LIN {X 0,Y 351.097,Z 362.91,A -85,B 0,C 180,E1 -17556.898,E2 -17556.898} C_VEL
LIN {X 0,Y 348.285,Z 360.251,A -85,B 0,C 180,E1 -17558.664,E2 -17558.664} C_VEL
LIN {X 0,Y 346.12,Z 358.177,A -85,B 0,C 180,E1 -17559.821,E2 -17559.821} C_VEL
LIN {X 0,Y 342.771,Z 355.678,A -85,B 0,C 180,E1 -17561.154,E2 -17561.154} C_VEL
LIN {X 0,Y 338.579,Z 351.959,A -85,B 0,C 180,E1 -17562.731,E2 -17562.731} C_VEL
LIN {X 0,Y 335.792,Z 349.388,A -85,B 0,C 180,E1 -17563.695,E2 -17563.695} C_VEL
LIN {X 0,Y 331.401,Z 345.387,A -85,B 0,C 180,E1 -17565.057,E2 -17565.057} C_VEL
LIN {X 0,Y 325.553,Z 339.743,A -85,B 0,C 180,E1 -17566.706,E2 -17566.706} C_VEL
LIN {X 0,Y 318.538,Z 332.574,A -85,B 0,C 180,E1 -17568.462,E2 -17568.462} C_VEL
LIN {X 0,Y 312.151,Z 325.702,A -85,B 0,C 180,E1 -17569.9,E2 -17569.9} C_VEL
LIN {X 0,Y 303.087,Z 315.131,A -85,B 0,C 180,E1 -17571.777,E2 -17571.777} C_VEL
LIN {X 0,Y 294.903,Z 304.725,A -85,B 0,C 180,E1 -17573.408,E2 -17573.408} C_VEL
LIN {X 0,Y 288.383,Z 294.709,A -85,B 0,C 180,E1 -17574.719,E2 -17574.719} C_VEL
LIN {X 0,Y 283.758,Z 285.694,A -85,B 0,C 180,E1 -17575.657,E2 -17575.657} C_VEL
LIN {X 0,Y 277.541,Z 272.57,A -85,B 0,C 180,E1 -17576.757,E2 -17576.757} C_VEL
LIN {X 0,Y 277.287,Z 271.445,A -85,B 0,C 180,E1 -17576.818,E2 -17576.818} C_VEL
LIN {X 0,Y 277.223,Z 271.454,A -85,B 0,C 180,E1 -17580.487,E2 -17580.487} C_VEL
LIN {X 0,Y 277.2,Z 271.458,A -85,B 0,C 180,E1 -17583.902,E2 -17583.902} C_VEL
LIN {X 0,Y 277.232,Z 271.452,A -85,B 0,C 180,E1 -17587.474,E2 -17587.474} C_VEL
LIN {X 0,Y 277.222,Z 271.452,A -85,B 0,C 180,E1 -17591.233,E2 -17591.233} C_VEL
LIN {X 0,Y 277.247,Z 271.449,A -85,B 0,C 180,E1 -17595.216,E2 -17595.216} C_VEL
LIN {X 0,Y 277.258,Z 271.45,A -85,B 0,C 180,E1 -17599.502,E2 -17599.502} C_VEL
LIN {X 0,Y 277.25,Z 271.448,A -85,B 0,C 180,E1 -17602.541,E2 -17602.541} C_VEL
LIN {X 0,Y 277.222,Z 271.451,A -85,B 0,C 180,E1 -17606.113,E2 -17606.113} C_VEL
LIN {X 0,Y 277.233,Z 271.452,A -85,B 0,C 180,E1 -17609.547,E2 -17609.547} C_VEL
LIN {X 0,Y 277.329,Z 271.44,A -85,B 0,C 180,E1 -17612.872,E2 -17612.872} C_VEL
LIN {X 0,Y 277.272,Z 271.443,A -85,B 0,C 180,E1 -17616.085,E2 -17616.085} C_VEL
LIN {X 0,Y 277.297,Z 271.441,A -85,B 0,C 180,E1 -17620.773,E2 -17620.773} C_VEL
LIN {X 0,Y 277.393,Z 271.428,A -85,B 0,C 180,E1 -17625.333,E2 -17625.333} C_VEL
LIN {X 0,Y 277.444,Z 271.421,A -85,B 0,C 180,E1 -17629.796,E2 -17629.796} C_VEL
LIN {X 0,Y 277.604,Z 271.406,A -85,B 0,C 180,E1 -17632.737,E2 -17632.737} C_VEL
LIN {X 0,Y 277.799,Z 271.368,A -85,B 0,C 180,E1 -17638.559,E2 -17638.559} C_VEL
LIN {X 0,Y 277.806,Z 271.376,A -85,B 0,C 180,E1 -17641.458,E2 -17641.458} C_VEL
LIN {X 0,Y 277.598,Z 271.404,A -85,B 0,C 180,E1 -17647.28,E2 -17647.28} C_VEL
LIN {X 0,Y 277.455,Z 271.425,A -85,B 0,C 180,E1 -17650.221,E2 -17650.221} C_VEL
LIN {X 0,Y 277.375,Z 271.433,A -85,B 0,C 180,E1 -17654.685,E2 -17654.685} C_VEL
LIN {X 0,Y 277.283,Z 271.445,A -85,B 0,C 180,E1 -17659.246,E2 -17659.246} C_VEL
LIN {X 0,Y 277.263,Z 271.448,A -85,B 0,C 180,E1 -17663.934,E2 -17663.934} C_VEL
LIN {X 0,Y 277.221,Z 271.451,A -85,B 0,C 180,E1 -17666.268,E2 -17666.268} C_VEL
LIN {X 0,Y 276.55,Z 271.54,A -85,B 0,C 180,E1 -17667.481,E2 -17667.481} C_VEL
LIN {X 0,Y 273.663,Z 271.899,A -85,B 0,C 180,E1 -17669.456,E2 -17669.456} C_VEL
LIN {X 0,Y 271.269,Z 272.403,A -85,B 0,C 180,E1 -17671.059,E2 -17671.059} C_VEL
LIN {X 0,Y 270.324,Z 272.925,A -85,B 0,C 180,E1 -17672.299,E2 -17672.299} C_VEL
LIN {X 0,Y 270.291,Z 273.131,A -85,B 0,C 180,E1 -17672.718,E2 -17672.718} C_VEL
LIN {X 0,Y 270.597,Z 275.334,A -85,B 0,C 180,E1 -17676.689,E2 -17676.689} C_VEL
LIN {X 0,Y 271.058,Z 278.164,A -85,B 0,C 180,E1 -17681.245,E2 -17681.245} C_VEL
LIN {X 0,Y 271.419,Z 281.232,A -85,B 0,C 180,E1 -17685.644,E2 -17685.644} C_VEL
LIN {X 0,Y 271.327,Z 283.569,A -85,B 0,C 180,E1 -17688.701,E2 -17688.701} C_VEL
LIN {X 0,Y 270.949,Z 285.847,A -85,B 0,C 180,E1 -17691.5,E2 -17691.5} C_VEL
LIN {X 0,Y 270.368,Z 288.968,A -85,B 0,C 180,E1 -17695.12,E2 -17695.12} C_VEL
LIN {X 0,Y 269.734,Z 292.721,A -85,B 0,C 180,E1 -17699.308,E2 -17699.308} C_VEL
LIN {X 0,Y 269.233,Z 295.826,A -85,B 0,C 180,E1 -17702.634,E2 -17702.634} C_VEL
LIN {X 0,Y 270.907,Z 301.981,A -85,B 0,C 180,E1 -17703.108,E2 -17703.108} C_VEL
LIN {X 0,Y 273.793,Z 313.364,A -85,B 0,C 180,E1 -17704.128,E2 -17704.128} C_VEL
LIN {X 0,Y 275.705,Z 322.952,A -85,B 0,C 180,E1 -17705.113,E2 -17705.113} C_VEL
LIN {X 0,Y 277,Z 333.021,A -85,B 0,C 180,E1 -17706.288,E2 -17706.288} C_VEL
LIN {X 0,Y 277.683,Z 342.384,A -85,B 0,C 180,E1 -17707.542,E2 -17707.542} C_VEL
LIN {X 0,Y 277.852,Z 346.126,A -85,B 0,C 180,E1 -17708.094,E2 -17708.094} C_VEL
LIN {X 0,Y 275.725,Z 357.626,A -85,B 0,C 180,E1 -17709.873,E2 -17709.873} C_VEL
LIN {X 0,Y 274.037,Z 366.483,A -85,B 0,C 180,E1 -17711.622,E2 -17711.622} C_VEL
LIN {X 0,Y 272.809,Z 372.974,A -85,B 0,C 180,E1 -17713.153,E2 -17713.153} C_VEL
LIN {X 0,Y 271.496,Z 379.514,A -85,B 0,C 180,E1 -17714.998,E2 -17714.998} C_VEL
LIN {X 0,Y 270.527,Z 384.016,A -85,B 0,C 180,E1 -17716.479,E2 -17716.479} C_VEL
LIN {X 0,Y 269.512,Z 389.513,A -85,B 0,C 180,E1 -17718.722,E2 -17718.722} C_VEL
LIN {X 0,Y 268.8,Z 393.843,A -85,B 0,C 180,E1 -17720.975,E2 -17720.975} C_VEL
LIN {X 0,Y 268.481,Z 396.213,A -85,B 0,C 180,E1 -17722.479,E2 -17722.479} C_VEL
LIN {X 0,Y 268.229,Z 398.793,A -85,B 0,C 180,E1 -17724.713,E2 -17724.713} C_VEL
LIN {X 0,Y 268.184,Z 400.47,A -85,B 0,C 180,E1 -17726.996,E2 -17726.996} C_VEL
LIN {X 0,Y 268.192,Z 401.061,A -85,B 0,C 180,E1 -17728.498,E2 -17728.498} C_VEL
LIN {X 0,Y 268.192,Z 401.061,A -85,B 0,C 180,E1 -17731.502,E2 -17731.502} C_VEL
LIN {X 0,Y 268.184,Z 400.47,A -85,B 0,C 180,E1 -17733.004,E2 -17733.004} C_VEL
LIN {X 0,Y 268.31,Z 398.017,A -85,B 0,C 180,E1 -17736.014,E2 -17736.014} C_VEL
LIN {X 0,Y 268.618,Z 395.061,A -85,B 0,C 180,E1 -17738.273,E2 -17738.273} C_VEL
LIN {X 0,Y 269.258,Z 391.069,A -85,B 0,C 180,E1 -17740.527,E2 -17740.527} C_VEL
LIN {X 0,Y 270.136,Z 385.933,A -85,B 0,C 180,E1 -17742.776,E2 -17742.776} C_VEL
LIN {X 0,Y 271.233,Z 380.67,A -85,B 0,C 180,E1 -17744.633,E2 -17744.633} C_VEL
LIN {X 0,Y 272.49,Z 374.349,A -85,B 0,C 180,E1 -17746.481,E2 -17746.481} C_VEL
LIN {X 0,Y 273.898,Z 367.698,A -85,B 0,C 180,E1 -17748.099,E2 -17748.099} C_VEL
LIN {X 0,Y 275.325,Z 359.545,A -85,B 0,C 180,E1 -17749.768,E2 -17749.768} C_VEL
LIN {X 0,Y 276.982,Z 351.016,A -85,B 0,C 180,E1 -17751.196,E2 -17751.196} C_VEL
LIN {X 0,Y 277.855,Z 346.126,A -85,B 0,C 180,E1 -17751.905,E2 -17751.905} C_VEL
LIN {X 0,Y 277.327,Z 336.813,A -85,B 0,C 180,E1 -17753.227,E2 -17753.227} C_VEL
LIN {X 0,Y 276.285,Z 326.665,A -85,B 0,C 180,E1 -17754.465,E2 -17754.465} C_VEL
LIN {X 0,Y 274.542,Z 316.92,A -85,B 0,C 180,E1 -17755.519,E2 -17755.519} C_VEL
LIN {X 0,Y 272.191,Z 306.812,A -85,B 0,C 180,E1 -17756.473,E2 -17756.473} C_VEL
LIN {X 0,Y 269.34,Z 296.803,A -85,B 0,C 180,E1 -17757.293,E2 -17757.293} C_VEL
LIN {X 0,Y 269.233,Z 295.84,A -85,B 0,C 180,E1 -17757.351,E2 -17757.351} C_VEL
LIN {X 0,Y 269.789,Z 292.071,A -85,B 0,C 180,E1 -17761.399,E2 -17761.399} C_VEL
LIN {X 0,Y 270.376,Z 288.938,A -85,B 0,C 180,E1 -17764.879,E2 -17764.879} C_VEL
LIN {X 0,Y 271.024,Z 285.471,A -85,B 0,C 180,E1 -17768.918,E2 -17768.918} C_VEL
LIN {X 0,Y 271.38,Z 282.742,A -85,B 0,C 180,E1 -17772.324,E2 -17772.324} C_VEL
LIN {X 0,Y 271.423,Z 281.192,A -85,B 0,C 180,E1 -17774.355,E2 -17774.355} C_VEL
LIN {X 0,Y 271.058,Z 278.155,A -85,B 0,C 180,E1 -17778.755,E2 -17778.755} C_VEL
LIN {X 0,Y 270.59,Z 275.327,A -85,B 0,C 180,E1 -17783.31,E2 -17783.31} C_VEL
LIN {X 0,Y 270.343,Z 273.321,A -85,B 0,C 180,E1 -17786.904,E2 -17786.904} C_VEL
LIN {X 0,Y 270.187,Z 272.33,A -85,B 0,C 180,E1 -17789.134,E2 -17789.134} C_VEL
LIN {X 0,Y 270.198,Z 272.33,A -85,B 0,C 180,E1 -17792.171,E2 -17792.171} C_VEL
LIN {X 0,Y 270.191,Z 272.331,A -85,B 0,C 180,E1 -17795.557,E2 -17795.557} C_VEL
LIN {X 0,Y 270.226,Z 272.328,A -85,B 0,C 180,E1 -17800.231,E2 -17800.231} C_VEL
LIN {X 0,Y 270.342,Z 272.309,A -85,B 0,C 180,E1 -17804.924,E2 -17804.924} C_VEL
LIN {X 0,Y 270.387,Z 272.304,A -85,B 0,C 180,E1 -17809.509,E2 -17809.509} C_VEL
LIN {X 0,Y 270.561,Z 272.281,A -85,B 0,C 180,E1 -17812.529,E2 -17812.529} C_VEL
LIN {X 0,Y 270.77,Z 272.253,A -85,B 0,C 180,E1 -17818.504,E2 -17818.504} C_VEL
LIN {X 0,Y 270.765,Z 272.242,A -85,B 0,C 180,E1 -17821.479,E2 -17821.479} C_VEL
LIN {X 0,Y 270.563,Z 272.285,A -85,B 0,C 180,E1 -17827.453,E2 -17827.453} C_VEL
LIN {X 0,Y 270.397,Z 272.299,A -85,B 0,C 180,E1 -17830.473,E2 -17830.473} C_VEL
LIN {X 0,Y 270.351,Z 272.306,A -85,B 0,C 180,E1 -17835.058,E2 -17835.058} C_VEL
LIN {X 0,Y 270.237,Z 272.317,A -85,B 0,C 180,E1 -17839.75,E2 -17839.75} C_VEL
LIN {X 0,Y 270.213,Z 272.325,A -85,B 0,C 180,E1 -17844.58,E2 -17844.58} C_VEL
LIN {X 0,Y 270.245,Z 272.32,A -85,B 0,C 180,E1 -17847.9,E2 -17847.9} C_VEL
LIN {X 0,Y 270.154,Z 272.332,A -85,B 0,C 180,E1 -17851.34,E2 -17851.34} C_VEL
LIN {X 0,Y 270.182,Z 272.33,A -85,B 0,C 180,E1 -17854.895,E2 -17854.895} C_VEL
LIN {X 0,Y 270.188,Z 272.331,A -85,B 0,C 180,E1 -17858.709,E2 -17858.709} C_VEL
LIN {X 0,Y 270.192,Z 272.329,A -85,B 0,C 180,E1 -17862.539,E2 -17862.539} C_VEL
LIN {X 0,Y 270.191,Z 272.328,A -85,B 0,C 180,E1 -17866.729,E2 -17866.729} C_VEL
LIN {X 0,Y 270.203,Z 272.325,A -85,B 0,C 180,E1 -17869.44,E2 -17869.44} C_VEL
LIN {X 0,Y 270.198,Z 272.328,A -85,B 0,C 180,E1 -17873.719,E2 -17873.719} C_VEL
LIN {X 0,Y 270.155,Z 272.332,A -85,B 0,C 180,E1 -17876.887,E2 -17876.887} C_VEL
LIN {X 0,Y 270.147,Z 272.335,A -85,B 0,C 180,E1 -17880.377,E2 -17880.377} C_VEL
LIN {X 0,Y 270.244,Z 272.323,A -85,B 0,C 180,E1 -17882.432,E2 -17882.432} C_VEL
LIN {X 0,Y 271.191,Z 275.041,A -85,B 0,C 180,E1 -17882.63,E2 -17882.63} C_VEL
LIN {X 0,Y 277.134,Z 287.397,A -85,B 0,C 180,E1 -17883.752,E2 -17883.752} C_VEL
LIN {X 0,Y 281.702,Z 297.031,A -85,B 0,C 180,E1 -17884.796,E2 -17884.796} C_VEL
LIN {X 0,Y 287.454,Z 306.253,A -85,B 0,C 180,E1 -17886.06,E2 -17886.06} C_VEL
LIN {X 0,Y 294.959,Z 316.48,A -85,B 0,C 180,E1 -17887.706,E2 -17887.706} C_VEL
LIN {X 0,Y 304.263,Z 327.414,A -85,B 0,C 180,E1 -17889.728,E2 -17889.728} C_VEL
LIN {X 0,Y 312.75,Z 336.664,A -85,B 0,C 180,E1 -17891.664,E2 -17891.664} C_VEL
LIN {X 0,Y 318.182,Z 342.223,A -85,B 0,C 180,E1 -17893.002,E2 -17893.002} C_VEL
LIN {X 0,Y 324.333,Z 348.16,A -85,B 0,C 180,E1 -17894.656,E2 -17894.656} C_VEL
LIN {X 0,Y 330.14,Z 353.561,A -85,B 0,C 180,E1 -17896.458,E2 -17896.458} C_VEL
LIN {X 0,Y 334.126,Z 357.349,A -85,B 0,C 180,E1 -17897.858,E2 -17897.858} C_VEL
LIN {X 0,Y 338.742,Z 361.057,A -85,B 0,C 180,E1 -17899.606,E2 -17899.606} C_VEL
LIN {X 0,Y 341.574,Z 363.402,A -85,B 0,C 180,E1 -17900.908,E2 -17900.908} C_VEL
LIN {X 0,Y 345.018,Z 366.712,A -85,B 0,C 180,E1 -17902.98,E2 -17902.98} C_VEL
LIN {X 0,Y 346.829,Z 368.073,A -85,B 0,C 180,E1 -17904.185,E2 -17904.185} C_VEL
LIN {X 0,Y 348.425,Z 369.044,A -85,B 0,C 180,E1 -17905.372,E2 -17905.372} C_VEL
LIN {X 0,Y 349.812,Z 369.646,A -85,B 0,C 180,E1 -17906.545,E2 -17906.545} C_VEL
LIN {X 0,Y 350.894,Z 370,A -85,B 0,C 180,E1 -17907.704,E2 -17907.704} C_VEL
LIN {X 0,Y 351.655,Z 370.14,A -85,B 0,C 180,E1 -17908.855,E2 -17908.855} C_VEL
LIN {X 0,Y 351.924,Z 370.171,A -85,B 0,C 180,E1 -17910,E2 -17910} C_VEL
LIN {X 0,Y 351.449,Z 370.117,A -85,B 0,C 180,E1 -17911.444,E2 -17911.444} C_VEL
LIN {X 0,Y 350.893,Z 369.986,A -85,B 0,C 180,E1 -17912.296,E2 -17912.296} C_VEL
LIN {X 0,Y 349.809,Z 369.639,A -85,B 0,C 180,E1 -17913.455,E2 -17913.455} C_VEL
LIN {X 0,Y 348.421,Z 369.058,A -85,B 0,C 180,E1 -17914.628,E2 -17914.628} C_VEL
LIN {X 0,Y 346.308,Z 367.73,A -85,B 0,C 180,E1 -17916.158,E2 -17916.158} C_VEL
LIN {X 0,Y 343.076,Z 364.884,A -85,B 0,C 180,E1 -17918.244,E2 -17918.244} C_VEL
LIN {X 0,Y 340.826,Z 362.661,A -85,B 0,C 180,E1 -17919.495,E2 -17919.495} C_VEL
LIN {X 0,Y 336.651,Z 359.474,A -85,B 0,C 180,E1 -17921.187,E2 -17921.187} C_VEL
LIN {X 0,Y 331.755,Z 355.007,A -85,B 0,C 180,E1 -17923.019,E2 -17923.019} C_VEL
LIN {X 0,Y 326.763,Z 350.61,A -85,B 0,C 180,E1 -17924.608,E2 -17924.608} C_VEL
LIN {X 0,Y 321.747,Z 345.628,A -85,B 0,C 180,E1 -17926.072,E2 -17926.072} C_VEL
LIN {X 0,Y 315.363,Z 339.315,A -85,B 0,C 180,E1 -17927.729,E2 -17927.729} C_VEL
LIN {X 0,Y 309.544,Z 333.151,A -85,B 0,C 180,E1 -17929.091,E2 -17929.091} C_VEL
LIN {X 0,Y 301.027,Z 323.692,A -85,B 0,C 180,E1 -17930.985,E2 -17930.985} C_VEL
LIN {X 0,Y 291.898,Z 312.497,A -85,B 0,C 180,E1 -17932.964,E2 -17932.964} C_VEL
LIN {X 0,Y 285.429,Z 303.26,A -85,B 0,C 180,E1 -17934.379,E2 -17934.379} C_VEL
LIN {X 0,Y 279.999,Z 293.639,A -85,B 0,C 180,E1 -17935.6,E2 -17935.6} C_VEL
LIN {X 0,Y 273.951,Z 280.6,A -85,B 0,C 180,E1 -17936.882,E2 -17936.882} C_VEL
LIN {X 0,Y 270.431,Z 273.312,A -85,B 0,C 180,E1 -17937.505,E2 -17937.505} C_VEL
LIN {X 0,Y 270.232,Z 272.325,A -85,B 0,C 180,E1 -17937.598,E2 -17937.598} C_VEL
LIN {X 0,Y 270.136,Z 272.335,A -85,B 0,C 180,E1 -17941.354,E2 -17941.354} C_VEL
LIN {X 0,Y 270.156,Z 272.332,A -85,B 0,C 180,E1 -17944.911,E2 -17944.911} C_VEL
LIN {X 0,Y 270.179,Z 272.329,A -85,B 0,C 180,E1 -17948.724,E2 -17948.724} C_VEL
LIN {X 0,Y 270.188,Z 272.327,A -85,B 0,C 180,E1 -17952.554,E2 -17952.554} C_VEL
LIN {X 0,Y 270.193,Z 272.327,A -85,B 0,C 180,E1 -17956.744,E2 -17956.744} C_VEL
LIN {X 0,Y 270.21,Z 272.327,A -85,B 0,C 180,E1 -17959.455,E2 -17959.455} C_VEL
LIN {X 0,Y 270.222,Z 272.325,A -85,B 0,C 180,E1 -17963.73,E2 -17963.73} C_VEL
LIN {X 0,Y 270.173,Z 272.33,A -85,B 0,C 180,E1 -17966.901,E2 -17966.901} C_VEL
LIN {X 0,Y 270.199,Z 272.326,A -85,B 0,C 180,E1 -17970.395,E2 -17970.395} C_VEL
LIN {X 0,Y 270.233,Z 272.32,A -85,B 0,C 180,E1 -17973.772,E2 -17973.772} C_VEL
LIN {X 0,Y 270.186,Z 272.331,A -85,B 0,C 180,E1 -17977.045,E2 -17977.045} C_VEL
LIN {X 0,Y 270.237,Z 272.317,A -85,B 0,C 180,E1 -17980.25,E2 -17980.25} C_VEL
LIN {X 0,Y 270.351,Z 272.306,A -85,B 0,C 180,E1 -17984.942,E2 -17984.942} C_VEL
LIN {X 0,Y 270.397,Z 272.299,A -85,B 0,C 180,E1 -17989.527,E2 -17989.527} C_VEL
LIN {X 0,Y 270.563,Z 272.285,A -85,B 0,C 180,E1 -17992.547,E2 -17992.547} C_VEL
LIN {X 0,Y 270.765,Z 272.242,A -85,B 0,C 180,E1 -17998.521,E2 -17998.521} C_VEL
LIN {X 0,Y 270.77,Z 272.253,A -85,B 0,C 180,E1 -18001.496,E2 -18001.496} C_VEL
LIN {X 0,Y 270.561,Z 272.282,A -85,B 0,C 180,E1 -18007.471,E2 -18007.471} C_VEL
LIN {X 0,Y 270.387,Z 272.304,A -85,B 0,C 180,E1 -18010.491,E2 -18010.491} C_VEL
LIN {X 0,Y 270.342,Z 272.309,A -85,B 0,C 180,E1 -18015.076,E2 -18015.076} C_VEL
LIN {X 0,Y 270.226,Z 272.327,A -85,B 0,C 180,E1 -18019.769,E2 -18019.769} C_VEL
LIN {X 0,Y 270.191,Z 272.327,A -85,B 0,C 180,E1 -18024.443,E2 -18024.443} C_VEL
LIN {X 0,Y 270.195,Z 272.33,A -85,B 0,C 180,E1 -18027.925,E2 -18027.925} C_VEL
LIN {X 0,Y 270.191,Z 272.433,A -85,B 0,C 180,E1 -18031.355,E2 -18031.355} C_VEL
LIN {X 0,Y 270.291,Z 273.131,A -85,B 0,C 180,E1 -18032.718,E2 -18032.718} C_VEL
LIN {X 0,Y 269.756,Z 273.889,A -85,B 0,C 180,E1 -18033.954,E2 -18033.954} C_VEL
LIN {X 0,Y 267.033,Z 275.456,A -85,B 0,C 180,E1 -18035.963,E2 -18035.963} C_VEL
LIN {X 0,Y 264.722,Z 276.769,A -85,B 0,C 180,E1 -18037.595,E2 -18037.595} C_VEL
LIN {X 0,Y 263.823,Z 277.672,A -85,B 0,C 180,E1 -18038.861,E2 -18038.861} C_VEL
LIN {X 0,Y 263.803,Z 277.94,A -85,B 0,C 180,E1 -18039.289,E2 -18039.289} C_VEL
LIN {X 0,Y 264.055,Z 279.533,A -85,B 0,C 180,E1 -18041.822,E2 -18041.822} C_VEL
LIN {X 0,Y 264.374,Z 282.305,A -85,B 0,C 180,E1 -18045.879,E2 -18045.879} C_VEL
LIN {X 0,Y 264.297,Z 284.143,A -85,B 0,C 180,E1 -18048.335,E2 -18048.335} C_VEL
LIN {X 0,Y 264.042,Z 285.878,A -85,B 0,C 180,E1 -18050.534,E2 -18050.534} C_VEL
LIN {X 0,Y 263.457,Z 288.799,A -85,B 0,C 180,E1 -18054.065,E2 -18054.065} C_VEL
LIN {X 0,Y 262.842,Z 291.894,A -85,B 0,C 180,E1 -18057.672,E2 -18057.672} C_VEL
LIN {X 0,Y 262.33,Z 295.013,A -85,B 0,C 180,E1 -18061.169,E2 -18061.169} C_VEL
LIN {X 0,Y 262.229,Z 295.648,A -85,B 0,C 180,E1 -18061.865,E2 -18061.865} C_VEL
LIN {X 0,Y 263.016,Z 298.737,A -85,B 0,C 180,E1 -18062.082,E2 -18062.082} C_VEL
LIN {X 0,Y 266.723,Z 312.289,A -85,B 0,C 180,E1 -18063.32,E2 -18063.32} C_VEL
LIN {X 0,Y 268.985,Z 323.726,A -85,B 0,C 180,E1 -18064.55,E2 -18064.55} C_VEL
LIN {X 0,Y 270.154,Z 332.334,A -85,B 0,C 180,E1 -18065.59,E2 -18065.59} C_VEL
LIN {X 0,Y 270.841,Z 341.367,A -85,B 0,C 180,E1 -18066.824,E2 -18066.824} C_VEL
LIN {X 0,Y 271.037,Z 347.266,A -85,B 0,C 180,E1 -18067.715,E2 -18067.715} C_VEL
LIN {X 0,Y 269.059,Z 357.414,A -85,B 0,C 180,E1 -18069.352,E2 -18069.352} C_VEL
LIN {X 0,Y 267.533,Z 365.254,A -85,B 0,C 180,E1 -18070.91,E2 -18070.91} C_VEL
LIN {X 0,Y 266.011,Z 372.762,A -85,B 0,C 180,E1 -18072.709,E2 -18072.709} C_VEL
LIN {X 0,Y 264.63,Z 379.302,A -85,B 0,C 180,E1 -18074.599,E2 -18074.599} C_VEL
LIN {X 0,Y 263.61,Z 383.804,A -85,B 0,C 180,E1 -18076.117,E2 -18076.117} C_VEL
LIN {X 0,Y 262.515,Z 389.3,A -85,B 0,C 180,E1 -18078.417,E2 -18078.417} C_VEL
LIN {X 0,Y 261.769,Z 393.631,A -85,B 0,C 180,E1 -18080.73,E2 -18080.73} C_VEL
LIN {X 0,Y 261.41,Z 396.001,A -85,B 0,C 180,E1 -18082.275,E2 -18082.275} C_VEL
LIN {X 0,Y 261.148,Z 398.736,A -85,B 0,C 180,E1 -18084.77,E2 -18084.77} C_VEL
LIN {X 0,Y 261.081,Z 400.258,A -85,B 0,C 180,E1 -18086.914,E2 -18086.914} C_VEL
LIN {X 0,Y 261.098,Z 400.85,A -85,B 0,C 180,E1 -18088.458,E2 -18088.458} C_VEL
LIN {X 0,Y 261.098,Z 400.85,A -85,B 0,C 180,E1 -18091.542,E2 -18091.542} C_VEL
LIN {X 0,Y 261.082,Z 400.258,A -85,B 0,C 180,E1 -18093.086,E2 -18093.086} C_VEL
LIN {X 0,Y 261.245,Z 397.805,A -85,B 0,C 180,E1 -18096.177,E2 -18096.177} C_VEL
LIN {X 0,Y 261.577,Z 394.849,A -85,B 0,C 180,E1 -18098.498,E2 -18098.498} C_VEL
LIN {X 0,Y 262.249,Z 390.857,A -85,B 0,C 180,E1 -18100.812,E2 -18100.812} C_VEL
LIN {X 0,Y 263.187,Z 385.721,A -85,B 0,C 180,E1 -18103.119,E2 -18103.119} C_VEL
LIN {X 0,Y 264.34,Z 380.457,A -85,B 0,C 180,E1 -18105.024,E2 -18105.024} C_VEL
LIN {X 0,Y 265.668,Z 374.137,A -85,B 0,C 180,E1 -18106.917,E2 -18106.917} C_VEL
LIN {X 0,Y 266.992,Z 368.186,A -85,B 0,C 180,E1 -18108.413,E2 -18108.413} C_VEL
LIN {X 0,Y 268.263,Z 361.253,A -85,B 0,C 180,E1 -18109.912,E2 -18109.912} C_VEL
LIN {X 0,Y 269.888,Z 353.073,A -85,B 0,C 180,E1 -18111.38,E2 -18111.38} C_VEL
LIN {X 0,Y 271.036,Z 347.266,A -85,B 0,C 180,E1 -18112.285,E2 -18112.285} C_VEL
LIN {X 0,Y 270.587,Z 337.402,A -85,B 0,C 180,E1 -18113.74,E2 -18113.74} C_VEL
LIN {X 0,Y 269.502,Z 326.882,A -85,B 0,C 180,E1 -18115.078,E2 -18115.078} C_VEL
LIN {X 0,Y 267.762,Z 317.114,A -85,B 0,C 180,E1 -18116.179,E2 -18116.179} C_VEL
LIN {X 0,Y 265.26,Z 306.595,A -85,B 0,C 180,E1 -18117.22,E2 -18117.22} C_VEL
LIN {X 0,Y 262.272,Z 296.17,A -85,B 0,C 180,E1 -18118.108,E2 -18118.108} C_VEL
LIN {X 0,Y 262.227,Z 295.617,A -85,B 0,C 180,E1 -18118.169,E2 -18118.169} C_VEL
LIN {X 0,Y 262.704,Z 292.95,A -85,B 0,C 180,E1 -18121.109,E2 -18121.109} C_VEL
LIN {X 0,Y 263.173,Z 290.304,A -85,B 0,C 180,E1 -18124.111,E2 -18124.111} C_VEL
LIN {X 0,Y 263.763,Z 287.175,A -85,B 0,C 180,E1 -18127.794,E2 -18127.794} C_VEL
LIN {X 0,Y 264.295,Z 284.115,A -85,B 0,C 180,E1 -18131.665,E2 -18131.665} C_VEL
LIN {X 0,Y 264.382,Z 282.301,A -85,B 0,C 180,E1 -18134.123,E2 -18134.123} C_VEL
LIN {X 0,Y 264.082,Z 279.455,A -85,B 0,C 180,E1 -18138.284,E2 -18138.284} C_VEL
LIN {X 0,Y 263.659,Z 277.055,A -85,B 0,C 180,E1 -18142.179,E2 -18142.179} C_VEL
LIN {X 0,Y 263.38,Z 274.957,A -85,B 0,C 180,E1 -18145.911,E2 -18145.911} C_VEL
LIN {X 0,Y 263.123,Z 273.21,A -85,B 0,C 180,E1 -18149.495,E2 -18149.495} C_VEL
LIN {X 0,Y 263.122,Z 273.212,A -85,B 0,C 180,E1 -18152.987,E2 -18152.987} C_VEL
LIN {X 0,Y 263.124,Z 273.215,A -85,B 0,C 180,E1 -18156.373,E2 -18156.373} C_VEL
LIN {X 0,Y 263.214,Z 273.2,A -85,B 0,C 180,E1 -18159.681,E2 -18159.681} C_VEL
LIN {X 0,Y 263.292,Z 273.189,A -85,B 0,C 180,E1 -18164.51,E2 -18164.51} C_VEL
LIN {X 0,Y 263.332,Z 273.182,A -85,B 0,C 180,E1 -18169.224,E2 -18169.224} C_VEL
LIN {X 0,Y 263.525,Z 273.159,A -85,B 0,C 180,E1 -18172.329,E2 -18172.329} C_VEL
LIN {X 0,Y 263.733,Z 273.129,A -85,B 0,C 180,E1 -18178.464,E2 -18178.464} C_VEL
LIN {X 0,Y 263.729,Z 273.117,A -85,B 0,C 180,E1 -18181.518,E2 -18181.518} C_VEL
LIN {X 0,Y 263.525,Z 273.159,A -85,B 0,C 180,E1 -18187.654,E2 -18187.654} C_VEL
LIN {X 0,Y 263.336,Z 273.179,A -85,B 0,C 180,E1 -18190.757,E2 -18190.757} C_VEL
LIN {X 0,Y 263.293,Z 273.186,A -85,B 0,C 180,E1 -18195.471,E2 -18195.471} C_VEL
LIN {X 0,Y 263.217,Z 273.191,A -85,B 0,C 180,E1 -18200.3,E2 -18200.3} C_VEL
LIN {X 0,Y 263.167,Z 273.201,A -85,B 0,C 180,E1 -18205.284,E2 -18205.284} C_VEL
LIN {X 0,Y 263.152,Z 273.207,A -85,B 0,C 180,E1 -18208.721,E2 -18208.721} C_VEL
LIN {X 0,Y 263.103,Z 273.211,A -85,B 0,C 180,E1 -18212.28,E2 -18212.28} C_VEL
LIN {X 0,Y 263.155,Z 273.204,A -85,B 0,C 180,E1 -18215.97,E2 -18215.97} C_VEL
LIN {X 0,Y 263.124,Z 273.208,A -85,B 0,C 180,E1 -18219.855,E2 -18219.855} C_VEL
LIN {X 0,Y 263.152,Z 273.206,A -85,B 0,C 180,E1 -18223.962,E2 -18223.962} C_VEL
LIN {X 0,Y 263.129,Z 273.209,A -85,B 0,C 180,E1 -18228.109,E2 -18228.109} C_VEL
LIN {X 0,Y 263.132,Z 273.21,A -85,B 0,C 180,E1 -18232.099,E2 -18232.099} C_VEL
LIN {X 0,Y 263.105,Z 273.213,A -85,B 0,C 180,E1 -18235.879,E2 -18235.879} C_VEL
LIN {X 0,Y 263.093,Z 273.214,A -85,B 0,C 180,E1 -18239.5,E2 -18239.5} C_VEL
LIN {X 0,Y 263.151,Z 273.207,A -85,B 0,C 180,E1 -18241.629,E2 -18241.629} C_VEL
LIN {X 0,Y 264.193,Z 276.077,A -85,B 0,C 180,E1 -18241.866,E2 -18241.866} C_VEL
LIN {X 0,Y 270.028,Z 287.992,A -85,B 0,C 180,E1 -18243.027,E2 -18243.027} C_VEL
LIN {X 0,Y 274.899,Z 298.832,A -85,B 0,C 180,E1 -18244.24,E2 -18244.24} C_VEL
LIN {X 0,Y 280.144,Z 308.035,A -85,B 0,C 180,E1 -18245.534,E2 -18245.534} C_VEL
LIN {X 0,Y 287.124,Z 317.874,A -85,B 0,C 180,E1 -18247.19,E2 -18247.19} C_VEL
LIN {X 0,Y 295.12,Z 327.693,A -85,B 0,C 180,E1 -18249.071,E2 -18249.071} C_VEL
LIN {X 0,Y 305.558,Z 339.141,A -85,B 0,C 180,E1 -18251.546,E2 -18251.546} C_VEL
LIN {X 0,Y 312.927,Z 346.66,A -85,B 0,C 180,E1 -18253.368,E2 -18253.368} C_VEL
LIN {X 0,Y 318.62,Z 352.081,A -85,B 0,C 180,E1 -18254.924,E2 -18254.924} C_VEL
LIN {X 0,Y 322.578,Z 355.933,A -85,B 0,C 180,E1 -18256.134,E2 -18256.134} C_VEL
LIN {X 0,Y 326.946,Z 359.876,A -85,B 0,C 180,E1 -18257.587,E2 -18257.587} C_VEL
LIN {X 0,Y 330.691,Z 363.155,A -85,B 0,C 180,E1 -18258.973,E2 -18258.973} C_VEL
LIN {X 0,Y 334.725,Z 366.265,A -85,B 0,C 180,E1 -18260.625,E2 -18260.625} C_VEL
LIN {X 0,Y 338.555,Z 369.968,A -85,B 0,C 180,E1 -18262.845,E2 -18262.845} C_VEL
LIN {X 0,Y 340.411,Z 371.44,A -85,B 0,C 180,E1 -18264.075,E2 -18264.075} C_VEL
LIN {X 0,Y 342.066,Z 372.452,A -85,B 0,C 180,E1 -18265.286,E2 -18265.286} C_VEL
LIN {X 0,Y 343.52,Z 373.131,A -85,B 0,C 180,E1 -18266.481,E2 -18266.481} C_VEL
LIN {X 0,Y 344.676,Z 373.556,A -85,B 0,C 180,E1 -18267.663,E2 -18267.663} C_VEL
LIN {X 0,Y 345.503,Z 373.744,A -85,B 0,C 180,E1 -18268.834,E2 -18268.834} C_VEL
LIN {X 0,Y 345.811,Z 373.784,A -85,B 0,C 180,E1 -18270,E2 -18270} C_VEL
LIN {X 0,Y 345.503,Z 373.73,A -85,B 0,C 180,E1 -18271.166,E2 -18271.166} C_VEL
LIN {X 0,Y 344.611,Z 373.535,A -85,B 0,C 180,E1 -18272.397,E2 -18272.397} C_VEL
LIN {X 0,Y 343.519,Z 373.131,A -85,B 0,C 180,E1 -18273.519,E2 -18273.519} C_VEL
LIN {X 0,Y 342.064,Z 372.471,A -85,B 0,C 180,E1 -18274.714,E2 -18274.714} C_VEL
LIN {X 0,Y 339.49,Z 370.775,A -85,B 0,C 180,E1 -18276.537,E2 -18276.537} C_VEL
LIN {X 0,Y 336.525,Z 368.019,A -85,B 0,C 180,E1 -18278.406,E2 -18278.406} C_VEL
LIN {X 0,Y 334.018,Z 365.72,A -85,B 0,C 180,E1 -18279.69,E2 -18279.69} C_VEL
LIN {X 0,Y 328.876,Z 361.606,A -85,B 0,C 180,E1 -18281.712,E2 -18281.712} C_VEL
LIN {X 0,Y 324.766,Z 357.806,A -85,B 0,C 180,E1 -18283.189,E2 -18283.189} C_VEL
LIN {X 0,Y 319.718,Z 353.2,A -85,B 0,C 180,E1 -18284.757,E2 -18284.757} C_VEL
LIN {X 0,Y 314.616,Z 348.29,A -85,B 0,C 180,E1 -18286.187,E2 -18286.187} C_VEL
LIN {X 0,Y 308.165,Z 341.786,A -85,B 0,C 180,E1 -18287.832,E2 -18287.832} C_VEL
LIN {X 0,Y 300.459,Z 333.663,A -85,B 0,C 180,E1 -18289.661,E2 -18289.661} C_VEL
LIN {X 0,Y 291.499,Z 323.371,A -85,B 0,C 180,E1 -18291.785,E2 -18291.785} C_VEL
LIN {X 0,Y 283.023,Z 312.363,A -85,B 0,C 180,E1 -18293.769,E2 -18293.769} C_VEL
LIN {X 0,Y 277.443,Z 303.564,A -85,B 0,C 180,E1 -18295.125,E2 -18295.125} C_VEL
LIN {X 0,Y 272.667,Z 294.101,A -85,B 0,C 180,E1 -18296.326,E2 -18296.326} C_VEL
LIN {X 0,Y 267.118,Z 281.719,A -85,B 0,C 180,E1 -18297.594,E2 -18297.594} C_VEL
LIN {X 0,Y 263.329,Z 274.154,A -85,B 0,C 180,E1 -18298.294,E2 -18298.294} C_VEL
LIN {X 0,Y 263.132,Z 273.21,A -85,B 0,C 180,E1 -18298.406,E2 -18298.406} C_VEL
LIN {X 0,Y 263.085,Z 273.215,A -85,B 0,C 180,E1 -18302.294,E2 -18302.294} C_VEL
LIN {X 0,Y 263.15,Z 273.205,A -85,B 0,C 180,E1 -18306.773,E2 -18306.773} C_VEL
LIN {X 0,Y 263.118,Z 273.211,A -85,B 0,C 180,E1 -18309.869,E2 -18309.869} C_VEL
LIN {X 0,Y 263.151,Z 273.206,A -85,B 0,C 180,E1 -18313.977,E2 -18313.977} C_VEL
LIN {X 0,Y 263.133,Z 273.207,A -85,B 0,C 180,E1 -18318.124,E2 -18318.124} C_VEL
LIN {X 0,Y 263.154,Z 273.204,A -85,B 0,C 180,E1 -18322.116,E2 -18322.116} C_VEL
LIN {X 0,Y 263.153,Z 273.204,A -85,B 0,C 180,E1 -18325.899,E2 -18325.899} C_VEL
LIN {X 0,Y 263.122,Z 273.21,A -85,B 0,C 180,E1 -18329.516,E2 -18329.516} C_VEL
LIN {X 0,Y 263.165,Z 273.206,A -85,B 0,C 180,E1 -18333.011,E2 -18333.011} C_VEL
LIN {X 0,Y 263.13,Z 273.206,A -85,B 0,C 180,E1 -18336.393,E2 -18336.393} C_VEL
LIN {X 0,Y 263.217,Z 273.191,A -85,B 0,C 180,E1 -18339.7,E2 -18339.7} C_VEL
LIN {X 0,Y 263.293,Z 273.186,A -85,B 0,C 180,E1 -18344.529,E2 -18344.529} C_VEL
LIN {X 0,Y 263.336,Z 273.179,A -85,B 0,C 180,E1 -18349.243,E2 -18349.243} C_VEL
LIN {X 0,Y 263.525,Z 273.159,A -85,B 0,C 180,E1 -18352.346,E2 -18352.346} C_VEL
LIN {X 0,Y 263.729,Z 273.117,A -85,B 0,C 180,E1 -18358.482,E2 -18358.482} C_VEL
LIN {X 0,Y 263.733,Z 273.129,A -85,B 0,C 180,E1 -18361.536,E2 -18361.536} C_VEL
LIN {X 0,Y 263.525,Z 273.159,A -85,B 0,C 180,E1 -18367.671,E2 -18367.671} C_VEL
LIN {X 0,Y 263.332,Z 273.182,A -85,B 0,C 180,E1 -18370.776,E2 -18370.776} C_VEL
LIN {X 0,Y 263.292,Z 273.189,A -85,B 0,C 180,E1 -18375.49,E2 -18375.49} C_VEL
LIN {X 0,Y 263.214,Z 273.197,A -85,B 0,C 180,E1 -18380.319,E2 -18380.319} C_VEL
LIN {X 0,Y 263.129,Z 273.21,A -85,B 0,C 180,E1 -18385.308,E2 -18385.308} C_VEL
LIN {X 0,Y 263.129,Z 273.211,A -85,B 0,C 180,E1 -18388.744,E2 -18388.744} C_VEL
LIN {X 0,Y 263.123,Z 273.212,A -85,B 0,C 180,E1 -18390.505,E2 -18390.505} C_VEL
LIN {X 0,Y 263.41,Z 275.017,A -85,B 0,C 180,E1 -18394.199,E2 -18394.199} C_VEL
LIN {X 0,Y 263.661,Z 277.058,A -85,B 0,C 180,E1 -18397.821,E2 -18397.821} C_VEL
LIN {X 0,Y 263.803,Z 277.94,A -85,B 0,C 180,E1 -18399.289,E2 -18399.289} C_VEL
LIN {X 0,Y 263.314,Z 278.812,A -85,B 0,C 180,E1 -18400.551,E2 -18400.551} C_VEL
LIN {X 0,Y 260.657,Z 280.533,A -85,B 0,C 180,E1 -18402.603,E2 -18402.603} C_VEL
LIN {X 0,Y 258.319,Z 281.98,A -85,B 0,C 180,E1 -18404.27,E2 -18404.27} C_VEL
LIN {X 0,Y 257.32,Z 283.005,A -85,B 0,C 180,E1 -18405.562,E2 -18405.562} C_VEL
LIN {X 0,Y 257.246,Z 283.321,A -85,B 0,C 180,E1 -18406,E2 -18406} C_VEL
LIN {X 0,Y 257.154,Z 285.531,A -85,B 0,C 180,E1 -18409.012,E2 -18409.012} C_VEL
LIN {X 0,Y 256.575,Z 288.612,A -85,B 0,C 180,E1 -18412.943,E2 -18412.943} C_VEL
LIN {X 0,Y 255.915,Z 291.717,A -85,B 0,C 180,E1 -18416.686,E2 -18416.686} C_VEL
LIN {X 0,Y 255.277,Z 295.445,A -85,B 0,C 180,E1 -18421.028,E2 -18421.028} C_VEL
LIN {X 0,Y 256.138,Z 298.689,A -85,B 0,C 180,E1 -18421.271,E2 -18421.271} C_VEL
LIN {X 0,Y 259.663,Z 311.352,A -85,B 0,C 180,E1 -18422.476,E2 -18422.476} C_VEL
LIN {X 0,Y 261.93,Z 322.375,A -85,B 0,C 180,E1 -18423.694,E2 -18423.694} C_VEL
LIN {X 0,Y 263.363,Z 332.093,A -85,B 0,C 180,E1 -18424.916,E2 -18424.916} C_VEL
LIN {X 0,Y 264.065,Z 341.374,A -85,B 0,C 180,E1 -18426.228,E2 -18426.228} C_VEL
LIN {X 0,Y 264.208,Z 348.315,A -85,B 0,C 180,E1 -18427.313,E2 -18427.313} C_VEL
LIN {X 0,Y 262.38,Z 357.201,A -85,B 0,C 180,E1 -18428.802,E2 -18428.802} C_VEL
LIN {X 0,Y 260.874,Z 364.719,A -85,B 0,C 180,E1 -18430.322,E2 -18430.322} C_VEL
LIN {X 0,Y 259.224,Z 372.586,A -85,B 0,C 180,E1 -18432.252,E2 -18432.252} C_VEL
LIN {X 0,Y 257.764,Z 379.09,A -85,B 0,C 180,E1 -18434.178,E2 -18434.178} C_VEL
LIN {X 0,Y 256.712,Z 383.593,A -85,B 0,C 180,E1 -18435.736,E2 -18435.736} C_VEL
LIN {X 0,Y 255.532,Z 389.088,A -85,B 0,C 180,E1 -18438.096,E2 -18438.096} C_VEL
LIN {X 0,Y 254.754,Z 393.419,A -85,B 0,C 180,E1 -18440.472,E2 -18440.472} C_VEL
LIN {X 0,Y 254.364,Z 395.789,A -85,B 0,C 180,E1 -18442.059,E2 -18442.059} C_VEL
LIN {X 0,Y 254.018,Z 398.984,A -85,B 0,C 180,E1 -18445.239,E2 -18445.239} C_VEL
LIN {X 0,Y 253.981,Z 400.047,A -85,B 0,C 180,E1 -18446.828,E2 -18446.828} C_VEL
LIN {X 0,Y 254.007,Z 400.639,A -85,B 0,C 180,E1 -18448.415,E2 -18448.415} C_VEL
LIN {X 0,Y 254.038,Z 400.795,A -85,B 0,C 180,E1 -18450,E2 -18450} C_VEL
LIN {X 0,Y 254.007,Z 400.639,A -85,B 0,C 180,E1 -18451.585,E2 -18451.585} C_VEL
LIN {X 0,Y 253.982,Z 400.047,A -85,B 0,C 180,E1 -18453.172,E2 -18453.172} C_VEL
LIN {X 0,Y 254.176,Z 397.593,A -85,B 0,C 180,E1 -18456.35,E2 -18456.35} C_VEL
LIN {X 0,Y 254.53,Z 394.637,A -85,B 0,C 180,E1 -18458.735,E2 -18458.735} C_VEL
LIN {X 0,Y 255.23,Z 390.644,A -85,B 0,C 180,E1 -18461.113,E2 -18461.113} C_VEL
LIN {X 0,Y 256.257,Z 385.509,A -85,B 0,C 180,E1 -18463.48,E2 -18463.48} C_VEL
LIN {X 0,Y 257.47,Z 380.246,A -85,B 0,C 180,E1 -18465.434,E2 -18465.434} C_VEL
LIN {X 0,Y 258.87,Z 373.925,A -85,B 0,C 180,E1 -18467.375,E2 -18467.375} C_VEL
LIN {X 0,Y 260.19,Z 367.972,A -85,B 0,C 180,E1 -18468.913,E2 -18468.913} C_VEL
LIN {X 0,Y 261.562,Z 361.041,A -85,B 0,C 180,E1 -18470.444,E2 -18470.444} C_VEL
LIN {X 0,Y 263.285,Z 352.861,A -85,B 0,C 180,E1 -18471.944,E2 -18471.944} C_VEL
LIN {X 0,Y 264.325,Z 347.05,A -85,B 0,C 180,E1 -18472.883,E2 -18472.883} C_VEL
LIN {X 0,Y 263.78,Z 337.197,A -85,B 0,C 180,E1 -18474.39,E2 -18474.39} C_VEL
LIN {X 0,Y 262.758,Z 327.155,A -85,B 0,C 180,E1 -18475.716,E2 -18475.716} C_VEL
LIN {X 0,Y 260.771,Z 316.365,A -85,B 0,C 180,E1 -18476.98,E2 -18476.98} C_VEL
LIN {X 0,Y 258.247,Z 305.915,A -85,B 0,C 180,E1 -18478.051,E2 -18478.051} C_VEL
LIN {X 0,Y 255.353,Z 296.272,A -85,B 0,C 180,E1 -18478.927,E2 -18478.927} C_VEL
LIN {X 0,Y 255.273,Z 295.447,A -85,B 0,C 180,E1 -18478.972,E2 -18478.972} C_VEL
LIN {X 0,Y 255.663,Z 293.19,A -85,B 0,C 180,E1 -18481.54,E2 -18481.54} C_VEL
LIN {X 0,Y 256.238,Z 290.121,A -85,B 0,C 180,E1 -18485.167,E2 -18485.167} C_VEL
LIN {X 0,Y 256.881,Z 286.995,A -85,B 0,C 180,E1 -18488.994,E2 -18488.994} C_VEL
LIN {X 0,Y 257.266,Z 284.401,A -85,B 0,C 180,E1 -18492.464,E2 -18492.464} C_VEL
LIN {X 0,Y 257.235,Z 282.43,A -85,B 0,C 180,E1 -18495.263,E2 -18495.263} C_VEL
LIN {X 0,Y 256.966,Z 280.01,A -85,B 0,C 180,E1 -18498.965,E2 -18498.965} C_VEL
LIN {X 0,Y 256.565,Z 277.666,A -85,B 0,C 180,E1 -18502.932,E2 -18502.932} C_VEL
LIN {X 0,Y 256.28,Z 275.635,A -85,B 0,C 180,E1 -18506.73,E2 -18506.73} C_VEL
LIN {X 0,Y 256.053,Z 274.092,A -85,B 0,C 180,E1 -18510.384,E2 -18510.384} C_VEL
LIN {X 0,Y 256.075,Z 274.091,A -85,B 0,C 180,E1 -18513.944,E2 -18513.944} C_VEL
LIN {X 0,Y 256.065,Z 274.091,A -85,B 0,C 180,E1 -18517.395,E2 -18517.395} C_VEL
LIN {X 0,Y 256.113,Z 274.084,A -85,B 0,C 180,E1 -18520.766,E2 -18520.766} C_VEL
LIN {X 0,Y 256.218,Z 274.072,A -85,B 0,C 180,E1 -18524.071,E2 -18524.071} C_VEL
LIN {X 0,Y 256.276,Z 274.061,A -85,B 0,C 180,E1 -18528.924,E2 -18528.924} C_VEL
LIN {X 0,Y 256.489,Z 274.037,A -85,B 0,C 180,E1 -18532.117,E2 -18532.117} C_VEL
LIN {X 0,Y 256.445,Z 274.039,A -85,B 0,C 180,E1 -18536.849,E2 -18536.849} C_VEL
LIN {X 0,Y 256.695,Z 274.006,A -85,B 0,C 180,E1 -18538.422,E2 -18538.422} C_VEL
LIN {X 0,Y 256.692,Z 273.992,A -85,B 0,C 180,E1 -18541.56,E2 -18541.56} C_VEL
LIN {X 0,Y 256.444,Z 274.037,A -85,B 0,C 180,E1 -18546.701,E2 -18546.701} C_VEL
LIN {X 0,Y 256.416,Z 274.042,A -85,B 0,C 180,E1 -18549.456,E2 -18549.456} C_VEL
LIN {X 0,Y 256.215,Z 274.065,A -85,B 0,C 180,E1 -18554.282,E2 -18554.282} C_VEL
LIN {X 0,Y 256.155,Z 274.077,A -85,B 0,C 180,E1 -18557.555,E2 -18557.555} C_VEL
LIN {X 0,Y 256.121,Z 274.08,A -85,B 0,C 180,E1 -18561.101,E2 -18561.101} C_VEL
LIN {X 0,Y 256.146,Z 274.075,A -85,B 0,C 180,E1 -18565.12,E2 -18565.12} C_VEL
LIN {X 0,Y 256.086,Z 274.085,A -85,B 0,C 180,E1 -18569.591,E2 -18569.591} C_VEL
LIN {X 0,Y 256.055,Z 274.088,A -85,B 0,C 180,E1 -18573.281,E2 -18573.281} C_VEL
LIN {X 0,Y 256.105,Z 274.082,A -85,B 0,C 180,E1 -18577.269,E2 -18577.269} C_VEL
LIN {X 0,Y 256.068,Z 274.087,A -85,B 0,C 180,E1 -18581.185,E2 -18581.185} C_VEL
LIN {X 0,Y 256.078,Z 274.087,A -85,B 0,C 180,E1 -18584.475,E2 -18584.475} C_VEL
LIN {X 0,Y 256.091,Z 274.084,A -85,B 0,C 180,E1 -18587.797,E2 -18587.797} C_VEL
LIN {X 0,Y 256.065,Z 274.088,A -85,B 0,C 180,E1 -18590.858,E2 -18590.858} C_VEL
LIN {X 0,Y 256.043,Z 274.091,A -85,B 0,C 180,E1 -18594.802,E2 -18594.802} C_VEL
LIN {X 0,Y 256.044,Z 274.091,A -85,B 0,C 180,E1 -18598.566,E2 -18598.566} C_VEL
LIN {X 0,Y 256.056,Z 274.109,A -85,B 0,C 180,E1 -18600.817,E2 -18600.817} C_VEL
LIN {X 0,Y 257.014,Z 276.836,A -85,B 0,C 180,E1 -18601.024,E2 -18601.024} C_VEL
LIN {X 0,Y 262.333,Z 287.24,A -85,B 0,C 180,E1 -18602.113,E2 -18602.113} C_VEL
LIN {X 0,Y 267.388,Z 299.066,A -85,B 0,C 180,E1 -18603.46,E2 -18603.46} C_VEL
LIN {X 0,Y 271.966,Z 308.03,A -85,B 0,C 180,E1 -18604.722,E2 -18604.722} C_VEL
LIN {X 0,Y 277.949,Z 317.476,A -85,B 0,C 180,E1 -18606.312,E2 -18606.312} C_VEL
LIN {X 0,Y 285.618,Z 327.28,A -85,B 0,C 180,E1 -18608.241,E2 -18608.241} C_VEL
LIN {X 0,Y 295.759,Z 338.768,A -85,B 0,C 180,E1 -18610.798,E2 -18610.798} C_VEL
LIN {X 0,Y 304.785,Z 347.955,A -85,B 0,C 180,E1 -18613.087,E2 -18613.087} C_VEL
LIN {X 0,Y 311.248,Z 354.223,A -85,B 0,C 180,E1 -18614.819,E2 -18614.819} C_VEL
LIN {X 0,Y 316.699,Z 359.422,A -85,B 0,C 180,E1 -18616.474,E2 -18616.474} C_VEL
LIN {X 0,Y 321.318,Z 363.626,A -85,B 0,C 180,E1 -18618.008,E2 -18618.008} C_VEL
LIN {X 0,Y 325.054,Z 366.784,A -85,B 0,C 180,E1 -18619.41,E2 -18619.41} C_VEL
LIN {X 0,Y 327.735,Z 368.864,A -85,B 0,C 180,E1 -18620.486,E2 -18620.486} C_VEL
LIN {X 0,Y 330.72,Z 371.679,A -85,B 0,C 180,E1 -18622.061,E2 -18622.061} C_VEL
LIN {X 0,Y 333.666,Z 374.215,A -85,B 0,C 180,E1 -18623.955,E2 -18623.955} C_VEL
LIN {X 0,Y 335.396,Z 375.332,A -85,B 0,C 180,E1 -18625.192,E2 -18625.192} C_VEL
LIN {X 0,Y 337.704,Z 376.458,A -85,B 0,C 180,E1 -18627.138,E2 -18627.138} C_VEL
LIN {X 0,Y 339.078,Z 376.861,A -85,B 0,C 180,E1 -18628.812,E2 -18628.812} C_VEL
LIN {X 0,Y 339.441,Z 376.914,A -85,B 0,C 180,E1 -18630,E2 -18630} C_VEL
LIN {X 0,Y 339.078,Z 376.849,A -85,B 0,C 180,E1 -18631.188,E2 -18631.188} C_VEL
LIN {X 0,Y 337.704,Z 376.468,A -85,B 0,C 180,E1 -18632.862,E2 -18632.862} C_VEL
LIN {X 0,Y 335.395,Z 375.354,A -85,B 0,C 180,E1 -18634.808,E2 -18634.808} C_VEL
LIN {X 0,Y 332.581,Z 373.341,A -85,B 0,C 180,E1 -18636.78,E2 -18636.78} C_VEL
LIN {X 0,Y 329.621,Z 370.556,A -85,B 0,C 180,E1 -18638.583,E2 -18638.583} C_VEL
LIN {X 0,Y 326.779,Z 368.138,A -85,B 0,C 180,E1 -18639.907,E2 -18639.907} C_VEL
LIN {X 0,Y 321.348,Z 363.62,A -85,B 0,C 180,E1 -18641.991,E2 -18641.991} C_VEL
LIN {X 0,Y 315.585,Z 358.418,A -85,B 0,C 180,E1 -18643.878,E2 -18643.878} C_VEL
LIN {X 0,Y 309.957,Z 352.983,A -85,B 0,C 180,E1 -18645.54,E2 -18645.54} C_VEL
LIN {X 0,Y 302.09,Z 345.262,A -85,B 0,C 180,E1 -18647.604,E2 -18647.604} C_VEL
LIN {X 0,Y 293.144,Z 335.93,A -85,B 0,C 180,E1 -18649.866,E2 -18649.866} C_VEL
LIN {X 0,Y 283.491,Z 324.782,A -85,B 0,C 180,E1 -18652.279,E2 -18652.279} C_VEL
LIN {X 0,Y 276.848,Z 315.843,A -85,B 0,C 180,E1 -18653.98,E2 -18653.98} C_VEL
LIN {X 0,Y 270.759,Z 305.867,A -85,B 0,C 180,E1 -18655.607,E2 -18655.607} C_VEL
LIN {X 0,Y 266.302,Z 296.415,A -85,B 0,C 180,E1 -18656.857,E2 -18656.857} C_VEL
LIN {X 0,Y 260.452,Z 283.235,A -85,B 0,C 180,E1 -18658.307,E2 -18658.307} C_VEL
LIN {X 0,Y 256.316,Z 275.277,A -85,B 0,C 180,E1 -18659.113,E2 -18659.113} C_VEL
LIN {X 0,Y 256.065,Z 274.089,A -85,B 0,C 180,E1 -18659.209,E2 -18659.209} C_VEL
LIN {X 0,Y 256.021,Z 274.094,A -85,B 0,C 180,E1 -18663.299,E2 -18663.299} C_VEL
LIN {X 0,Y 256.085,Z 274.086,A -85,B 0,C 180,E1 -18667.282,E2 -18667.282} C_VEL
LIN {X 0,Y 256.063,Z 274.088,A -85,B 0,C 180,E1 -18671.201,E2 -18671.201} C_VEL
LIN {X 0,Y 256.077,Z 274.085,A -85,B 0,C 180,E1 -18674.491,E2 -18674.491} C_VEL
LIN {X 0,Y 256.095,Z 274.086,A -85,B 0,C 180,E1 -18677.812,E2 -18677.812} C_VEL
LIN {X 0,Y 256.074,Z 274.087,A -85,B 0,C 180,E1 -18680.873,E2 -18680.873} C_VEL
LIN {X 0,Y 256.089,Z 274.084,A -85,B 0,C 180,E1 -18684.822,E2 -18684.822} C_VEL
LIN {X 0,Y 256.063,Z 274.087,A -85,B 0,C 180,E1 -18688.581,E2 -18688.581} C_VEL
LIN {X 0,Y 256.114,Z 274.081,A -85,B 0,C 180,E1 -18692.205,E2 -18692.205} C_VEL
LIN {X 0,Y 256.118,Z 274.079,A -85,B 0,C 180,E1 -18695.706,E2 -18695.706} C_VEL
LIN {X 0,Y 256.128,Z 274.077,A -85,B 0,C 180,E1 -18699.113,E2 -18699.113} C_VEL
LIN {X 0,Y 256.228,Z 274.066,A -85,B 0,C 180,E1 -18704.091,E2 -18704.091} C_VEL
LIN {X 0,Y 256.277,Z 274.059,A -85,B 0,C 180,E1 -18708.943,E2 -18708.943} C_VEL
LIN {X 0,Y 256.487,Z 274.035,A -85,B 0,C 180,E1 -18712.135,E2 -18712.135} C_VEL
LIN {X 0,Y 256.452,Z 274.023,A -85,B 0,C 180,E1 -18716.867,E2 -18716.867} C_VEL
LIN {X 0,Y 256.692,Z 273.992,A -85,B 0,C 180,E1 -18718.44,E2 -18718.44} C_VEL
LIN {X 0,Y 256.695,Z 274.006,A -85,B 0,C 180,E1 -18721.578,E2 -18721.578} C_VEL
LIN {X 0,Y 256.452,Z 274.041,A -85,B 0,C 180,E1 -18726.302,E2 -18726.302} C_VEL
LIN {X 0,Y 256.404,Z 274.046,A -85,B 0,C 180,E1 -18729.475,E2 -18729.475} C_VEL
LIN {X 0,Y 256.205,Z 274.072,A -85,B 0,C 180,E1 -18734.302,E2 -18734.302} C_VEL
LIN {X 0,Y 256.153,Z 274.079,A -85,B 0,C 180,E1 -18737.574,E2 -18737.574} C_VEL
LIN {X 0,Y 256.127,Z 274.08,A -85,B 0,C 180,E1 -18741.104,E2 -18741.104} C_VEL
LIN {X 0,Y 256.091,Z 274.085,A -85,B 0,C 180,E1 -18745.094,E2 -18745.094} C_VEL
LIN {X 0,Y 256.087,Z 274.088,A -85,B 0,C 180,E1 -18748.576,E2 -18748.576} C_VEL
LIN {X 0,Y 256.053,Z 274.093,A -85,B 0,C 180,E1 -18749.616,E2 -18749.616} C_VEL
LIN {X 0,Y 256.3,Z 275.631,A -85,B 0,C 180,E1 -18753.267,E2 -18753.267} C_VEL
LIN {X 0,Y 256.598,Z 277.878,A -85,B 0,C 180,E1 -18757.414,E2 -18757.414} C_VEL
LIN {X 0,Y 256.932,Z 280.029,A -85,B 0,C 180,E1 -18761.041,E2 -18761.041} C_VEL
LIN {X 0,Y 257.256,Z 282.809,A -85,B 0,C 180,E1 -18765.268,E2 -18765.268} C_VEL
LIN {X 0,Y 257.246,Z 283.321,A -85,B 0,C 180,E1 -18766,E2 -18766} C_VEL
LIN {X 0,Y 256.565,Z 284.333,A -85,B 0,C 180,E1 -18767.286,E2 -18767.286} C_VEL
LIN {X 0,Y 254.912,Z 285.466,A -85,B 0,C 180,E1 -18768.54,E2 -18768.54} C_VEL
LIN {X 0,Y 250.894,Z 287.786,A -85,B 0,C 180,E1 -18771.052,E2 -18771.052} C_VEL
LIN {X 0,Y 249.632,Z 288.905,A -85,B 0,C 180,E1 -18772.369,E2 -18772.369} C_VEL
LIN {X 0,Y 249.467,Z 289.266,A -85,B 0,C 180,E1 -18772.819,E2 -18772.819} C_VEL
LIN {X 0,Y 249.048,Z 291.539,A -85,B 0,C 180,E1 -18775.641,E2 -18775.641} C_VEL
LIN {X 0,Y 248.321,Z 295.227,A -85,B 0,C 180,E1 -18780.122,E2 -18780.122} C_VEL
LIN {X 0,Y 249.227,Z 298.601,A -85,B 0,C 180,E1 -18780.403,E2 -18780.403} C_VEL
LIN {X 0,Y 252.94,Z 311.65,A -85,B 0,C 180,E1 -18781.725,E2 -18781.725} C_VEL
LIN {X 0,Y 255.293,Z 323.272,A -85,B 0,C 180,E1 -18783.078,E2 -18783.078} C_VEL
LIN {X 0,Y 256.641,Z 332.425,A -85,B 0,C 180,E1 -18784.285,E2 -18784.285} C_VEL
LIN {X 0,Y 257.297,Z 341.385,A -85,B 0,C 180,E1 -18785.599,E2 -18785.599} C_VEL
LIN {X 0,Y 257.413,Z 349.245,A -85,B 0,C 180,E1 -18786.892,E2 -18786.892} C_VEL
LIN {X 0,Y 255.779,Z 356.99,A -85,B 0,C 180,E1 -18788.227,E2 -18788.227} C_VEL
LIN {X 0,Y 254.161,Z 364.503,A -85,B 0,C 180,E1 -18789.779,E2 -18789.779} C_VEL
LIN {X 0,Y 252.427,Z 372.514,A -85,B 0,C 180,E1 -18791.8,E2 -18791.8} C_VEL
LIN {X 0,Y 250.904,Z 378.878,A -85,B 0,C 180,E1 -18793.734,E2 -18793.734} C_VEL
LIN {X 0,Y 249.83,Z 383.381,A -85,B 0,C 180,E1 -18795.335,E2 -18795.335} C_VEL
LIN {X 0,Y 248.562,Z 388.876,A -85,B 0,C 180,E1 -18797.757,E2 -18797.757} C_VEL
LIN {X 0,Y 247.715,Z 393.207,A -85,B 0,C 180,E1 -18800.199,E2 -18800.199} C_VEL
LIN {X 0,Y 247.312,Z 395.577,A -85,B 0,C 180,E1 -18801.831,E2 -18801.831} C_VEL
LIN {X 0,Y 246.969,Z 398.653,A -85,B 0,C 180,E1 -18804.937,E2 -18804.937} C_VEL
LIN {X 0,Y 246.885,Z 399.835,A -85,B 0,C 180,E1 -18806.736,E2 -18806.736} C_VEL
LIN {X 0,Y 246.917,Z 400.428,A -85,B 0,C 180,E1 -18808.369,E2 -18808.369} C_VEL
LIN {X 0,Y 246.968,Z 400.585,A -85,B 0,C 180,E1 -18810,E2 -18810} C_VEL
LIN {X 0,Y 246.917,Z 400.428,A -85,B 0,C 180,E1 -18811.631,E2 -18811.631} C_VEL
LIN {X 0,Y 246.887,Z 399.835,A -85,B 0,C 180,E1 -18813.264,E2 -18813.264} C_VEL
LIN {X 0,Y 247.09,Z 397.381,A -85,B 0,C 180,E1 -18816.533,E2 -18816.533} C_VEL
LIN {X 0,Y 247.504,Z 394.426,A -85,B 0,C 180,E1 -18818.985,E2 -18818.985} C_VEL
LIN {X 0,Y 248.232,Z 390.431,A -85,B 0,C 180,E1 -18821.431,E2 -18821.431} C_VEL
LIN {X 0,Y 249.317,Z 385.296,A -85,B 0,C 180,E1 -18823.863,E2 -18823.863} C_VEL
LIN {X 0,Y 250.615,Z 380.034,A -85,B 0,C 180,E1 -18825.868,E2 -18825.868} C_VEL
LIN {X 0,Y 252.096,Z 373.714,A -85,B 0,C 180,E1 -18827.858,E2 -18827.858} C_VEL
LIN {X 0,Y 253.422,Z 367.759,A -85,B 0,C 180,E1 -18829.438,E2 -18829.438} C_VEL
LIN {X 0,Y 254.894,Z 360.828,A -85,B 0,C 180,E1 -18831.004,E2 -18831.004} C_VEL
LIN {X 0,Y 256.717,Z 352.65,A -85,B 0,C 180,E1 -18832.536,E2 -18832.536} C_VEL
LIN {X 0,Y 257.559,Z 348.1,A -85,B 0,C 180,E1 -18833.307,E2 -18833.307} C_VEL
LIN {X 0,Y 257.093,Z 338.137,A -85,B 0,C 180,E1 -18834.915,E2 -18834.915} C_VEL
LIN {X 0,Y 255.97,Z 327.423,A -85,B 0,C 180,E1 -18836.396,E2 -18836.396} C_VEL
LIN {X 0,Y 254.047,Z 316.721,A -85,B 0,C 180,E1 -18837.704,E2 -18837.704} C_VEL
LIN {X 0,Y 251.562,Z 306.532,A -85,B 0,C 180,E1 -18838.811,E2 -18838.811} C_VEL
LIN {X 0,Y 248.4,Z 295.911,A -85,B 0,C 180,E1 -18839.822,E2 -18839.822} C_VEL
LIN {X 0,Y 248.319,Z 295.232,A -85,B 0,C 180,E1 -18839.878,E2 -18839.878} C_VEL
LIN {X 0,Y 249.048,Z 291.445,A -85,B 0,C 180,E1 -18844.359,E2 -18844.359} C_VEL
LIN {X 0,Y 249.691,Z 288.383,A -85,B 0,C 180,E1 -18848.259,E2 -18848.259} C_VEL
LIN {X 0,Y 250.038,Z 286.588,A -85,B 0,C 180,E1 -18850.622,E2 -18850.622} C_VEL
LIN {X 0,Y 250.234,Z 284.834,A -85,B 0,C 180,E1 -18853.085,E2 -18853.085} C_VEL
LIN {X 0,Y 250.069,Z 282.259,A -85,B 0,C 180,E1 -18856.945,E2 -18856.945} C_VEL
LIN {X 0,Y 249.842,Z 280.569,A -85,B 0,C 180,E1 -18859.676,E2 -18859.676} C_VEL
LIN {X 0,Y 249.461,Z 278.287,A -85,B 0,C 180,E1 -18863.718,E2 -18863.718} C_VEL
LIN {X 0,Y 249.206,Z 276.21,A -85,B 0,C 180,E1 -18867.782,E2 -18867.782} C_VEL
LIN {X 0,Y 249.036,Z 274.966,A -85,B 0,C 180,E1 -18871.025,E2 -18871.025} C_VEL
LIN {X 0,Y 249.064,Z 274.965,A -85,B 0,C 180,E1 -18874.95,E2 -18874.95} C_VEL
LIN {X 0,Y 249.059,Z 274.965,A -85,B 0,C 180,E1 -18878.62,E2 -18878.62} C_VEL
LIN {X 0,Y 249.164,Z 274.948,A -85,B 0,C 180,E1 -18883.608,E2 -18883.608} C_VEL
LIN {X 0,Y 249.221,Z 274.941,A -85,B 0,C 180,E1 -18888.606,E2 -18888.606} C_VEL
LIN {X 0,Y 249.431,Z 274.917,A -85,B 0,C 180,E1 -18891.892,E2 -18891.892} C_VEL
LIN {X 0,Y 249.257,Z 274.935,A -85,B 0,C 180,E1 -18895.139,E2 -18895.139} C_VEL
LIN {X 0,Y 249.655,Z 274.883,A -85,B 0,C 180,E1 -18898.378,E2 -18898.378} C_VEL
LIN {X 0,Y 249.653,Z 274.867,A -85,B 0,C 180,E1 -18901.604,E2 -18901.604} C_VEL
LIN {X 0,Y 249.416,Z 274.913,A -85,B 0,C 180,E1 -18906.686,E2 -18906.686} C_VEL
LIN {X 0,Y 249.331,Z 274.923,A -85,B 0,C 180,E1 -18909.727,E2 -18909.727} C_VEL
LIN {X 0,Y 249.159,Z 274.945,A -85,B 0,C 180,E1 -18914.696,E2 -18914.696} C_VEL
LIN {X 0,Y 249.089,Z 274.956,A -85,B 0,C 180,E1 -18918.07,E2 -18918.07} C_VEL
LIN {X 0,Y 249.06,Z 274.961,A -85,B 0,C 180,E1 -18921.509,E2 -18921.509} C_VEL
LIN {X 0,Y 249.092,Z 274.954,A -85,B 0,C 180,E1 -18925.465,E2 -18925.465} C_VEL
LIN {X 0,Y 249.056,Z 274.962,A -85,B 0,C 180,E1 -18928.983,E2 -18928.983} C_VEL
LIN {X 0,Y 249.006,Z 274.968,A -85,B 0,C 180,E1 -18932.416,E2 -18932.416} C_VEL
LIN {X 0,Y 249.041,Z 274.963,A -85,B 0,C 180,E1 -18936.329,E2 -18936.329} C_VEL
LIN {X 0,Y 249.042,Z 274.964,A -85,B 0,C 180,E1 -18940.456,E2 -18940.456} C_VEL
LIN {X 0,Y 249.023,Z 274.965,A -85,B 0,C 180,E1 -18944.858,E2 -18944.858} C_VEL
LIN {X 0,Y 249.038,Z 274.961,A -85,B 0,C 180,E1 -18947.368,E2 -18947.368} C_VEL
LIN {X 0,Y 249.005,Z 274.968,A -85,B 0,C 180,E1 -18951.616,E2 -18951.616} C_VEL
LIN {X 0,Y 249,Z 274.969,A -85,B 0,C 180,E1 -18955.633,E2 -18955.633} C_VEL
LIN {X 0,Y 249.012,Z 275.037,A -85,B 0,C 180,E1 -18959.93,E2 -18959.93} C_VEL
LIN {X 0,Y 250.025,Z 277.863,A -85,B 0,C 180,E1 -18960.166,E2 -18960.166} C_VEL
LIN {X 0,Y 255.736,Z 288.924,A -85,B 0,C 180,E1 -18961.415,E2 -18961.415} C_VEL
LIN {X 0,Y 260.644,Z 300.522,A -85,B 0,C 180,E1 -18962.823,E2 -18962.823} C_VEL
LIN {X 0,Y 265.233,Z 310.357,A -85,B 0,C 180,E1 -18964.251,E2 -18964.251} C_VEL
LIN {X 0,Y 270.789,Z 319.484,A -85,B 0,C 180,E1 -18965.864,E2 -18965.864} C_VEL
LIN {X 0,Y 277.2,Z 328.245,A -85,B 0,C 180,E1 -18967.648,E2 -18967.648} C_VEL
LIN {X 0,Y 286.01,Z 338.396,A -85,B 0,C 180,E1 -18969.999,E2 -18969.999} C_VEL
LIN {X 0,Y 294.906,Z 347.629,A -85,B 0,C 180,E1 -18972.375,E2 -18972.375} C_VEL
LIN {X 0,Y 302.641,Z 355.009,A -85,B 0,C 180,E1 -18974.478,E2 -18974.478} C_VEL
LIN {X 0,Y 308.4,Z 360.396,A -85,B 0,C 180,E1 -18976.157,E2 -18976.157} C_VEL
LIN {X 0,Y 313.266,Z 364.757,A -85,B 0,C 180,E1 -18977.694,E2 -18977.694} C_VEL
LIN {X 0,Y 317.338,Z 368.427,A -85,B 0,C 180,E1 -18979.178,E2 -18979.178} C_VEL
LIN {X 0,Y 320.64,Z 371.047,A -85,B 0,C 180,E1 -18980.454,E2 -18980.454} C_VEL
LIN {X 0,Y 323.585,Z 373.645,A -85,B 0,C 180,E1 -18981.884,E2 -18981.884} C_VEL
LIN {X 0,Y 326.659,Z 376.373,A -85,B 0,C 180,E1 -18983.825,E2 -18983.825} C_VEL
LIN {X 0,Y 328.457,Z 377.665,A -85,B 0,C 180,E1 -18985.09,E2 -18985.09} C_VEL
LIN {X 0,Y 330.742,Z 378.89,A -85,B 0,C 180,E1 -18986.888,E2 -18986.888} C_VEL
LIN {X 0,Y 332.407,Z 379.467,A -85,B 0,C 180,E1 -18988.789,E2 -18988.789} C_VEL
LIN {X 0,Y 332.844,Z 379.527,A -85,B 0,C 180,E1 -18990,E2 -18990} C_VEL
LIN {X 0,Y 332.407,Z 379.456,A -85,B 0,C 180,E1 -18991.211,E2 -18991.211} C_VEL
LIN {X 0,Y 330.742,Z 378.881,A -85,B 0,C 180,E1 -18993.112,E2 -18993.112} C_VEL
LIN {X 0,Y 328.457,Z 377.679,A -85,B 0,C 180,E1 -18994.91,E2 -18994.91} C_VEL
LIN {X 0,Y 325.575,Z 375.488,A -85,B 0,C 180,E1 -18996.884,E2 -18996.884} C_VEL
LIN {X 0,Y 323.605,Z 373.656,A -85,B 0,C 180,E1 -18998.115,E2 -18998.115} C_VEL
LIN {X 0,Y 320.641,Z 371.034,A -85,B 0,C 180,E1 -18999.547,E2 -18999.547} C_VEL
LIN {X 0,Y 315.365,Z 366.681,A -85,B 0,C 180,E1 -19001.57,E2 -19001.57} C_VEL
LIN {X 0,Y 310.379,Z 362.229,A -85,B 0,C 180,E1 -19003.227,E2 -19003.227} C_VEL
LIN {X 0,Y 304.464,Z 356.626,A -85,B 0,C 180,E1 -19005.021,E2 -19005.021} C_VEL
LIN {X 0,Y 296.404,Z 349.066,A -85,B 0,C 180,E1 -19007.226,E2 -19007.226} C_VEL
LIN {X 0,Y 287.275,Z 339.764,A -85,B 0,C 180,E1 -19009.667,E2 -19009.667} C_VEL
LIN {X 0,Y 278.489,Z 329.799,A -85,B 0,C 180,E1 -19012.008,E2 -19012.008} C_VEL
LIN {X 0,Y 271.596,Z 320.719,A -85,B 0,C 180,E1 -19013.902,E2 -19013.902} C_VEL
LIN {X 0,Y 265.83,Z 311.366,A -85,B 0,C 180,E1 -19015.579,E2 -19015.579} C_VEL
LIN {X 0,Y 261.443,Z 302.547,A -85,B 0,C 180,E1 -19016.913,E2 -19016.913} C_VEL
LIN {X 0,Y 256.533,Z 290.736,A -85,B 0,C 180,E1 -19018.371,E2 -19018.371} C_VEL
LIN {X 0,Y 251.952,Z 281.342,A -85,B 0,C 180,E1 -19019.448,E2 -19019.448} C_VEL
LIN {X 0,Y 249.263,Z 276.154,A -85,B 0,C 180,E1 -19019.999,E2 -19019.999} C_VEL
LIN {X 0,Y 248.999,Z 274.97,A -85,B 0,C 180,E1 -19020.117,E2 -19020.117} C_VEL
LIN {X 0,Y 249,Z 274.969,A -85,B 0,C 180,E1 -19024.367,E2 -19024.367} C_VEL
LIN {X 0,Y 249.005,Z 274.968,A -85,B 0,C 180,E1 -19028.384,E2 -19028.384} C_VEL
LIN {X 0,Y 249.038,Z 274.961,A -85,B 0,C 180,E1 -19032.632,E2 -19032.632} C_VEL
LIN {X 0,Y 249.041,Z 274.963,A -85,B 0,C 180,E1 -19037.384,E2 -19037.384} C_VEL
LIN {X 0,Y 249.018,Z 274.967,A -85,B 0,C 180,E1 -19041.633,E2 -19041.633} C_VEL
LIN {X 0,Y 249.03,Z 274.964,A -85,B 0,C 180,E1 -19045.651,E2 -19045.651} C_VEL
LIN {X 0,Y 249.023,Z 274.967,A -85,B 0,C 180,E1 -19049.482,E2 -19049.482} C_VEL
LIN {X 0,Y 249.044,Z 274.963,A -85,B 0,C 180,E1 -19053.171,E2 -19053.171} C_VEL
LIN {X 0,Y 249.037,Z 274.963,A -85,B 0,C 180,E1 -19056.74,E2 -19056.74} C_VEL
LIN {X 0,Y 249.063,Z 274.954,A -85,B 0,C 180,E1 -19060.219,E2 -19060.219} C_VEL
LIN {X 0,Y 249.179,Z 274.943,A -85,B 0,C 180,E1 -19063.628,E2 -19063.628} C_VEL
LIN {X 0,Y 249.22,Z 274.941,A -85,B 0,C 180,E1 -19068.625,E2 -19068.625} C_VEL
LIN {X 0,Y 249.43,Z 274.913,A -85,B 0,C 180,E1 -19071.911,E2 -19071.911} C_VEL
LIN {X 0,Y 249.266,Z 274.928,A -85,B 0,C 180,E1 -19075.158,E2 -19075.158} C_VEL
LIN {X 0,Y 249.653,Z 274.867,A -85,B 0,C 180,E1 -19078.396,E2 -19078.396} C_VEL
LIN {X 0,Y 249.655,Z 274.883,A -85,B 0,C 180,E1 -19081.622,E2 -19081.622} C_VEL
LIN {X 0,Y 249.426,Z 274.916,A -85,B 0,C 180,E1 -19086.48,E2 -19086.48} C_VEL
LIN {X 0,Y 249.334,Z 274.928,A -85,B 0,C 180,E1 -19089.746,E2 -19089.746} C_VEL
LIN {X 0,Y 249.15,Z 274.949,A -85,B 0,C 180,E1 -19094.715,E2 -19094.715} C_VEL
LIN {X 0,Y 249.085,Z 274.959,A -85,B 0,C 180,E1 -19098.09,E2 -19098.09} C_VEL
LIN {X 0,Y 249.051,Z 274.965,A -85,B 0,C 180,E1 -19101.53,E2 -19101.53} C_VEL
LIN {X 0,Y 249.053,Z 274.964,A -85,B 0,C 180,E1 -19105.446,E2 -19105.446} C_VEL
LIN {X 0,Y 249.036,Z 274.967,A -85,B 0,C 180,E1 -19108.975,E2 -19108.975} C_VEL
LIN {X 0,Y 249.219,Z 276.302,A -85,B 0,C 180,E1 -19112.407,E2 -19112.407} C_VEL
LIN {X 0,Y 249.469,Z 278.289,A -85,B 0,C 180,E1 -19116.28,E2 -19116.28} C_VEL
LIN {X 0,Y 249.868,Z 280.749,A -85,B 0,C 180,E1 -19120.588,E2 -19120.588} C_VEL
LIN {X 0,Y 250.172,Z 283.282,A -85,B 0,C 180,E1 -19124.623,E2 -19124.623} C_VEL
LIN {X 0,Y 250.188,Z 285.366,A -85,B 0,C 180,E1 -19127.61,E2 -19127.61} C_VEL
LIN {X 0,Y 250.014,Z 286.902,A -85,B 0,C 180,E1 -19129.72,E2 -19129.72} C_VEL
LIN {X 0,Y 249.467,Z 289.266,A -85,B 0,C 180,E1 -19132.819,E2 -19132.819} C_VEL
LIN {X 0,Y 248.63,Z 290.036,A -85,B 0,C 180,E1 -19133.693,E2 -19133.693} C_VEL
LIN {X 0,Y 245.551,Z 291.416,A -85,B 0,C 180,E1 -19135.042,E2 -19135.042} C_VEL
LIN {X 0,Y 242.459,Z 292.768,A -85,B 0,C 180,E1 -19136.422,E2 -19136.422} C_VEL
LIN {X 0,Y 241.64,Z 293.537,A -85,B 0,C 180,E1 -19137.332,E2 -19137.332} C_VEL
LIN {X 0,Y 241.372,Z 295.182,A -85,B 0,C 180,E1 -19139.195,E2 -19139.195} C_VEL
LIN {X 0,Y 242.205,Z 298.229,A -85,B 0,C 180,E1 -19139.449,E2 -19139.449} C_VEL
LIN {X 0,Y 246.06,Z 311.273,A -85,B 0,C 180,E1 -19140.847,E2 -19140.847} C_VEL
LIN {X 0,Y 248.369,Z 322.256,A -85,B 0,C 180,E1 -19142.175,E2 -19142.175} C_VEL
LIN {X 0,Y 249.912,Z 332.428,A -85,B 0,C 180,E1 -19143.57,E2 -19143.57} C_VEL
LIN {X 0,Y 250.569,Z 341.406,A -85,B 0,C 180,E1 -19144.938,E2 -19144.938} C_VEL
LIN {X 0,Y 250.645,Z 350.169,A -85,B 0,C 180,E1 -19146.449,E2 -19146.449} C_VEL
LIN {X 0,Y 248.695,Z 358.697,A -85,B 0,C 180,E1 -19148.011,E2 -19148.011} C_VEL
LIN {X 0,Y 247.09,Z 365.919,A -85,B 0,C 180,E1 -19149.609,E2 -19149.609} C_VEL
LIN {X 0,Y 245.626,Z 372.442,A -85,B 0,C 180,E1 -19151.322,E2 -19151.322} C_VEL
LIN {X 0,Y 244.056,Z 378.665,A -85,B 0,C 180,E1 -19153.264,E2 -19153.264} C_VEL
LIN {X 0,Y 242.929,Z 383.169,A -85,B 0,C 180,E1 -19154.908,E2 -19154.908} C_VEL
LIN {X 0,Y 241.58,Z 388.663,A -85,B 0,C 180,E1 -19157.398,E2 -19157.398} C_VEL
LIN {X 0,Y 240.695,Z 392.995,A -85,B 0,C 180,E1 -19159.91,E2 -19159.91} C_VEL
LIN {X 0,Y 240.262,Z 395.365,A -85,B 0,C 180,E1 -19161.59,E2 -19161.59} C_VEL
LIN {X 0,Y 239.986,Z 397.168,A -85,B 0,C 180,E1 -19163.273,E2 -19163.273} C_VEL
LIN {X 0,Y 239.794,Z 399.624,A -85,B 0,C 180,E1 -19166.64,E2 -19166.64} C_VEL
LIN {X 0,Y 239.83,Z 400.217,A -85,B 0,C 180,E1 -19168.321,E2 -19168.321} C_VEL
LIN {X 0,Y 239.878,Z 400.374,A -85,B 0,C 180,E1 -19170,E2 -19170} C_VEL
LIN {X 0,Y 239.83,Z 400.217,A -85,B 0,C 180,E1 -19171.679,E2 -19171.679} C_VEL
LIN {X 0,Y 239.795,Z 399.624,A -85,B 0,C 180,E1 -19173.36,E2 -19173.36} C_VEL
LIN {X 0,Y 240.015,Z 397.169,A -85,B 0,C 180,E1 -19176.726,E2 -19176.726} C_VEL
LIN {X 0,Y 240.463,Z 394.213,A -85,B 0,C 180,E1 -19179.25,E2 -19179.25} C_VEL
LIN {X 0,Y 241.252,Z 390.219,A -85,B 0,C 180,E1 -19181.766,E2 -19181.766} C_VEL
LIN {X 0,Y 242.399,Z 385.084,A -85,B 0,C 180,E1 -19184.267,E2 -19184.267} C_VEL
LIN {X 0,Y 243.77,Z 379.822,A -85,B 0,C 180,E1 -19186.325,E2 -19186.325} C_VEL
LIN {X 0,Y 245.343,Z 373.503,A -85,B 0,C 180,E1 -19188.367,E2 -19188.367} C_VEL
LIN {X 0,Y 246.691,Z 367.546,A -85,B 0,C 180,E1 -19189.99,E2 -19189.99} C_VEL
LIN {X 0,Y 248.239,Z 360.616,A -85,B 0,C 180,E1 -19191.595,E2 -19191.595} C_VEL
LIN {X 0,Y 250.173,Z 352.439,A -85,B 0,C 180,E1 -19193.159,E2 -19193.159} C_VEL
LIN {X 0,Y 250.782,Z 349.03,A -85,B 0,C 180,E1 -19193.756,E2 -19193.756} C_VEL
LIN {X 0,Y 250.295,Z 336.968,A -85,B 0,C 180,E1 -19195.769,E2 -19195.769} C_VEL
LIN {X 0,Y 249.249,Z 327.705,A -85,B 0,C 180,E1 -19197.109,E2 -19197.109} C_VEL
LIN {X 0,Y 247.358,Z 317.129,A -85,B 0,C 180,E1 -19198.464,E2 -19198.464} C_VEL
LIN {X 0,Y 244.879,Z 307.048,A -85,B 0,C 180,E1 -19199.624,E2 -19199.624} C_VEL
LIN {X 0,Y 241.761,Z 297.116,A -85,B 0,C 180,E1 -19200.663,E2 -19200.663} C_VEL
LIN {X 0,Y 241.356,Z 295.018,A -85,B 0,C 180,E1 -19200.843,E2 -19200.843} C_VEL
LIN {X 0,Y 242.153,Z 291.26,A -85,B 0,C 180,E1 -19205.482,E2 -19205.482} C_VEL
LIN {X 0,Y 242.818,Z 288.193,A -85,B 0,C 180,E1 -19209.55,E2 -19209.55} C_VEL
LIN {X 0,Y 243.053,Z 286.67,A -85,B 0,C 180,E1 -19211.686,E2 -19211.686} C_VEL
LIN {X 0,Y 243.168,Z 285.15,A -85,B 0,C 180,E1 -19213.918,E2 -19213.918} C_VEL
LIN {X 0,Y 243.06,Z 283.616,A -85,B 0,C 180,E1 -19216.291,E2 -19216.291} C_VEL
LIN {X 0,Y 242.887,Z 282.083,A -85,B 0,C 180,E1 -19218.79,E2 -19218.79} C_VEL
LIN {X 0,Y 242.533,Z 279.982,A -85,B 0,C 180,E1 -19222.507,E2 -19222.507} C_VEL
LIN {X 0,Y 242.249,Z 277.894,A -85,B 0,C 180,E1 -19226.54,E2 -19226.54} C_VEL
LIN {X 0,Y 241.989,Z 276.034,A -85,B 0,C 180,E1 -19230.606,E2 -19230.606} C_VEL
LIN {X 0,Y 242.007,Z 275.845,A -85,B 0,C 180,E1 -19234.19,E2 -19234.19} C_VEL
LIN {X 0,Y 241.994,Z 275.847,A -85,B 0,C 180,E1 -19238.33,E2 -19238.33} C_VEL
LIN {X 0,Y 242.112,Z 275.826,A -85,B 0,C 180,E1 -19243.316,E2 -19243.316} C_VEL
LIN {X 0,Y 242.155,Z 275.823,A -85,B 0,C 180,E1 -19248.269,E2 -19248.269} C_VEL
LIN {X 0,Y 242.381,Z 275.794,A -85,B 0,C 180,E1 -19251.655,E2 -19251.655} C_VEL
LIN {X 0,Y 242.398,Z 275.79,A -85,B 0,C 180,E1 -19253.331,E2 -19253.331} C_VEL
LIN {X 0,Y 242.615,Z 275.76,A -85,B 0,C 180,E1 -19258.33,E2 -19258.33} C_VEL
LIN {X 0,Y 242.614,Z 275.742,A -85,B 0,C 180,E1 -19261.65,E2 -19261.65} C_VEL
LIN {X 0,Y 242.398,Z 275.789,A -85,B 0,C 180,E1 -19266.658,E2 -19266.658} C_VEL
LIN {X 0,Y 242.254,Z 275.804,A -85,B 0,C 180,E1 -19270.014,E2 -19270.014} C_VEL
LIN {X 0,Y 242.118,Z 275.822,A -85,B 0,C 180,E1 -19275.133,E2 -19275.133} C_VEL
LIN {X 0,Y 242.027,Z 275.836,A -85,B 0,C 180,E1 -19278.616,E2 -19278.616} C_VEL
LIN {X 0,Y 241.983,Z 275.841,A -85,B 0,C 180,E1 -19282.171,E2 -19282.171} C_VEL
LIN {X 0,Y 242.043,Z 275.831,A -85,B 0,C 180,E1 -19285.828,E2 -19285.828} C_VEL
LIN {X 0,Y 242.003,Z 275.839,A -85,B 0,C 180,E1 -19289.571,E2 -19289.571} C_VEL
LIN {X 0,Y 241.961,Z 275.843,A -85,B 0,C 180,E1 -19293.482,E2 -19293.482} C_VEL
LIN {X 0,Y 241.978,Z 275.842,A -85,B 0,C 180,E1 -19297.569,E2 -19297.569} C_VEL
LIN {X 0,Y 241.958,Z 275.846,A -85,B 0,C 180,E1 -19301.902,E2 -19301.902} C_VEL
LIN {X 0,Y 241.968,Z 275.844,A -85,B 0,C 180,E1 -19305.807,E2 -19305.807} C_VEL
LIN {X 0,Y 241.965,Z 275.846,A -85,B 0,C 180,E1 -19310.283,E2 -19310.283} C_VEL
LIN {X 0,Y 241.949,Z 275.848,A -85,B 0,C 180,E1 -19314.484,E2 -19314.484} C_VEL
LIN {X 0,Y 241.944,Z 275.848,A -85,B 0,C 180,E1 -19318.952,E2 -19318.952} C_VEL
LIN {X 0,Y 242.982,Z 278.756,A -85,B 0,C 180,E1 -19319.238,E2 -19319.238} C_VEL
LIN {X 0,Y 248.684,Z 289.587,A -85,B 0,C 180,E1 -19320.555,E2 -19320.555} C_VEL
LIN {X 0,Y 252.947,Z 299.522,A -85,B 0,C 180,E1 -19321.815,E2 -19321.815} C_VEL
LIN {X 0,Y 257.028,Z 309.352,A -85,B 0,C 180,E1 -19323.227,E2 -19323.227} C_VEL
LIN {X 0,Y 261.267,Z 317.6,A -85,B 0,C 180,E1 -19324.644,E2 -19324.644} C_VEL
LIN {X 0,Y 267.798,Z 327.644,A -85,B 0,C 180,E1 -19326.682,E2 -19326.682} C_VEL
LIN {X 0,Y 276.226,Z 338.013,A -85,B 0,C 180,E1 -19329.133,E2 -19329.133} C_VEL
LIN {X 0,Y 285.068,Z 347.295,A -85,B 0,C 180,E1 -19331.614,E2 -19331.614} C_VEL
LIN {X 0,Y 294.036,Z 355.752,A -85,B 0,C 180,E1 -19334.131,E2 -19334.131} C_VEL
LIN {X 0,Y 300.04,Z 361.08,A -85,B 0,C 180,E1 -19335.878,E2 -19335.878} C_VEL
LIN {X 0,Y 307.046,Z 367.268,A -85,B 0,C 180,E1 -19338.112,E2 -19338.112} C_VEL
LIN {X 0,Y 311.03,Z 370.799,A -85,B 0,C 180,E1 -19339.586,E2 -19339.586} C_VEL
LIN {X 0,Y 314.64,Z 373.72,A -85,B 0,C 180,E1 -19341.005,E2 -19341.005} C_VEL
LIN {X 0,Y 317.347,Z 376.087,A -85,B 0,C 180,E1 -19342.364,E2 -19342.364} C_VEL
LIN {X 0,Y 319.414,Z 377.924,A -85,B 0,C 180,E1 -19343.684,E2 -19343.684} C_VEL
LIN {X 0,Y 321.31,Z 379.412,A -85,B 0,C 180,E1 -19344.981,E2 -19344.981} C_VEL
LIN {X 0,Y 323.731,Z 380.807,A -85,B 0,C 180,E1 -19346.803,E2 -19346.803} C_VEL
LIN {X 0,Y 325.529,Z 381.466,A -85,B 0,C 180,E1 -19348.763,E2 -19348.763} C_VEL
LIN {X 0,Y 326.018,Z 381.531,A -85,B 0,C 180,E1 -19350,E2 -19350} C_VEL
LIN {X 0,Y 325.529,Z 381.457,A -85,B 0,C 180,E1 -19351.237,E2 -19351.237} C_VEL
LIN {X 0,Y 323.727,Z 380.804,A -85,B 0,C 180,E1 -19353.186,E2 -19353.186} C_VEL
LIN {X 0,Y 321.31,Z 379.403,A -85,B 0,C 180,E1 -19355.019,E2 -19355.019} C_VEL
LIN {X 0,Y 318.512,Z 377.152,A -85,B 0,C 180,E1 -19356.908,E2 -19356.908} C_VEL
LIN {X 0,Y 316.097,Z 374.987,A -85,B 0,C 180,E1 -19358.309,E2 -19358.309} C_VEL
LIN {X 0,Y 313.457,Z 372.755,A -85,B 0,C 180,E1 -19359.485,E2 -19359.485} C_VEL
LIN {X 0,Y 308.276,Z 368.38,A -85,B 0,C 180,E1 -19361.446,E2 -19361.446} C_VEL
LIN {X 0,Y 302.165,Z 363.019,A -85,B 0,C 180,E1 -19363.449,E2 -19363.449} C_VEL
LIN {X 0,Y 295.314,Z 356.908,A -85,B 0,C 180,E1 -19365.498,E2 -19365.498} C_VEL
LIN {X 0,Y 286.349,Z 348.53,A -85,B 0,C 180,E1 -19368.038,E2 -19368.038} C_VEL
LIN {X 0,Y 277.555,Z 339.435,A -85,B 0,C 180,E1 -19370.5,E2 -19370.5} C_VEL
LIN {X 0,Y 268.489,Z 328.516,A -85,B 0,C 180,E1 -19373.118,E2 -19373.118} C_VEL
LIN {X 0,Y 261.881,Z 318.622,A -85,B 0,C 180,E1 -19375.162,E2 -19375.162} C_VEL
LIN {X 0,Y 257.029,Z 309.317,A -85,B 0,C 180,E1 -19376.777,E2 -19376.777} C_VEL
LIN {X 0,Y 252.959,Z 299.521,A -85,B 0,C 180,E1 -19378.184,E2 -19378.184} C_VEL
LIN {X 0,Y 247.809,Z 287.809,A -85,B 0,C 180,E1 -19379.676,E2 -19379.676} C_VEL
LIN {X 0,Y 242.876,Z 278.539,A -85,B 0,C 180,E1 -19380.791,E2 -19380.791} C_VEL
LIN {X 0,Y 241.944,Z 275.848,A -85,B 0,C 180,E1 -19381.048,E2 -19381.048} C_VEL
LIN {X 0,Y 241.961,Z 275.847,A -85,B 0,C 180,E1 -19385.603,E2 -19385.603} C_VEL
LIN {X 0,Y 241.965,Z 275.846,A -85,B 0,C 180,E1 -19389.717,E2 -19389.717} C_VEL
LIN {X 0,Y 241.968,Z 275.844,A -85,B 0,C 180,E1 -19394.193,E2 -19394.193} C_VEL
LIN {X 0,Y 241.958,Z 275.846,A -85,B 0,C 180,E1 -19398.098,E2 -19398.098} C_VEL
LIN {X 0,Y 241.978,Z 275.842,A -85,B 0,C 180,E1 -19402.431,E2 -19402.431} C_VEL
LIN {X 0,Y 241.961,Z 275.843,A -85,B 0,C 180,E1 -19406.518,E2 -19406.518} C_VEL
LIN {X 0,Y 242.01,Z 275.839,A -85,B 0,C 180,E1 -19410.597,E2 -19410.597} C_VEL
LIN {X 0,Y 242.044,Z 275.831,A -85,B 0,C 180,E1 -19414.193,E2 -19414.193} C_VEL
LIN {X 0,Y 242.002,Z 275.839,A -85,B 0,C 180,E1 -19418.325,E2 -19418.325} C_VEL
LIN {X 0,Y 242.099,Z 275.826,A -85,B 0,C 180,E1 -19423.326,E2 -19423.326} C_VEL
LIN {X 0,Y 242.153,Z 275.822,A -85,B 0,C 180,E1 -19428.289,E2 -19428.289} C_VEL
LIN {X 0,Y 242.379,Z 275.791,A -85,B 0,C 180,E1 -19431.674,E2 -19431.674} C_VEL
LIN {X 0,Y 242.227,Z 275.805,A -85,B 0,C 180,E1 -19435.017,E2 -19435.017} C_VEL
LIN {X 0,Y 242.614,Z 275.742,A -85,B 0,C 180,E1 -19438.35,E2 -19438.35} C_VEL
LIN {X 0,Y 242.615,Z 275.76,A -85,B 0,C 180,E1 -19441.67,E2 -19441.67} C_VEL
LIN {X 0,Y 242.398,Z 275.791,A -85,B 0,C 180,E1 -19446.669,E2 -19446.669} C_VEL
LIN {X 0,Y 242.262,Z 275.81,A -85,B 0,C 180,E1 -19450.033,E2 -19450.033} C_VEL
LIN {X 0,Y 242.109,Z 275.827,A -85,B 0,C 180,E1 -19455.154,E2 -19455.154} C_VEL
LIN {X 0,Y 242.024,Z 275.837,A -85,B 0,C 180,E1 -19458.637,E2 -19458.637} C_VEL
LIN {X 0,Y 241.981,Z 275.843,A -85,B 0,C 180,E1 -19462.192,E2 -19462.192} C_VEL
LIN {X 0,Y 241.997,Z 275.841,A -85,B 0,C 180,E1 -19465.834,E2 -19465.834} C_VEL
LIN {X 0,Y 242.006,Z 276.12,A -85,B 0,C 180,E1 -19469.593,E2 -19469.593} C_VEL
LIN {X 0,Y 242.258,Z 277.915,A -85,B 0,C 180,E1 -19473.458,E2 -19473.458} C_VEL
LIN {X 0,Y 242.536,Z 279.986,A -85,B 0,C 180,E1 -19477.492,E2 -19477.492} C_VEL
LIN {X 0,Y 242.916,Z 282.405,A -85,B 0,C 180,E1 -19481.725,E2 -19481.725} C_VEL
LIN {X 0,Y 243.191,Z 285.158,A -85,B 0,C 180,E1 -19486.087,E2 -19486.087} C_VEL
LIN {X 0,Y 243.01,Z 287.023,A -85,B 0,C 180,E1 -19488.769,E2 -19488.769} C_VEL
LIN {X 0,Y 242.456,Z 289.779,A -85,B 0,C 180,E1 -19492.504,E2 -19492.504} C_VEL
LIN {X 0,Y 241.799,Z 292.87,A -85,B 0,C 180,E1 -19496.48,E2 -19496.48} C_VEL
LIN {X 0,Y 241.64,Z 293.537,A -85,B 0,C 180,E1 -19497.332,E2 -19497.332} C_VEL
LIN {X 0,Y 241.509,Z 295.031,A -85,B 0,C 180,E1 -19498.138,E2 -19498.138} C_VEL
LIN {X 0,Y 241.385,Z 297.62,A -85,B 0,C 180,E1 -19498.79,E2 -19498.79} C_VEL
LIN {X 0,Y 241.188,Z 302.665,A -85,B 0,C 180,E1 -19499.518,E2 -19499.518} C_VEL
LIN {X 0,Y 241.132,Z 318.872,A -85,B 0,C 180,E1 -19500.911,E2 -19500.911} C_VEL
LIN {X 0,Y 241.356,Z 320.781,A -85,B 0,C 180,E1 -19501.148,E2 -19501.148} C_VEL
LIN {X 0,Y 243.005,Z 331.365,A -85,B 0,C 180,E1 -19502.64,E2 -19502.64} C_VEL
LIN {X 0,Y 243.83,Z 341.165,A -85,B 0,C 180,E1 -19504.192,E2 -19504.192} C_VEL
LIN {X 0,Y 243.998,Z 349.952,A -85,B 0,C 180,E1 -19505.767,E2 -19505.767} C_VEL
LIN {X 0,Y 242.121,Z 358.485,A -85,B 0,C 180,E1 -19507.381,E2 -19507.381} C_VEL
LIN {X 0,Y 240.414,Z 365.707,A -85,B 0,C 180,E1 -19509.017,E2 -19509.017} C_VEL
LIN {X 0,Y 239,Z 371.785,A -85,B 0,C 180,E1 -19510.64,E2 -19510.64} C_VEL
LIN {X 0,Y 237.223,Z 378.453,A -85,B 0,C 180,E1 -19512.767,E2 -19512.767} C_VEL
LIN {X 0,Y 236.041,Z 382.956,A -85,B 0,C 180,E1 -19514.457,E2 -19514.457} C_VEL
LIN {X 0,Y 234.618,Z 388.451,A -85,B 0,C 180,E1 -19517.017,E2 -19517.017} C_VEL
LIN {X 0,Y 233.662,Z 392.782,A -85,B 0,C 180,E1 -19519.603,E2 -19519.603} C_VEL
LIN {X 0,Y 233.231,Z 395.153,A -85,B 0,C 180,E1 -19521.335,E2 -19521.335} C_VEL
LIN {X 0,Y 232.922,Z 396.957,A -85,B 0,C 180,E1 -19523.068,E2 -19523.068} C_VEL
LIN {X 0,Y 232.706,Z 399.412,A -85,B 0,C 180,E1 -19526.537,E2 -19526.537} C_VEL
LIN {X 0,Y 232.744,Z 400.006,A -85,B 0,C 180,E1 -19528.27,E2 -19528.27} C_VEL
LIN {X 0,Y 232.791,Z 400.163,A -85,B 0,C 180,E1 -19530,E2 -19530} C_VEL
LIN {X 0,Y 232.744,Z 400.006,A -85,B 0,C 180,E1 -19531.73,E2 -19531.73} C_VEL
LIN {X 0,Y 232.774,Z 398.607,A -85,B 0,C 180,E1 -19534.822,E2 -19534.822} C_VEL
LIN {X 0,Y 232.942,Z 396.957,A -85,B 0,C 180,E1 -19536.931,E2 -19536.931} C_VEL
LIN {X 0,Y 233.441,Z 394.002,A -85,B 0,C 180,E1 -19539.531,E2 -19539.531} C_VEL
LIN {X 0,Y 234.283,Z 390.007,A -85,B 0,C 180,E1 -19542.121,E2 -19542.121} C_VEL
LIN {X 0,Y 235.498,Z 384.872,A -85,B 0,C 180,E1 -19544.694,E2 -19544.694} C_VEL
LIN {X 0,Y 236.937,Z 379.609,A -85,B 0,C 180,E1 -19546.81,E2 -19546.81} C_VEL
LIN {X 0,Y 238.602,Z 373.291,A -85,B 0,C 180,E1 -19548.905,E2 -19548.905} C_VEL
LIN {X 0,Y 239.981,Z 367.333,A -85,B 0,C 180,E1 -19550.574,E2 -19550.574} C_VEL
LIN {X 0,Y 241.635,Z 360.404,A -85,B 0,C 180,E1 -19552.216,E2 -19552.216} C_VEL
LIN {X 0,Y 243.633,Z 352.226,A -85,B 0,C 180,E1 -19553.819,E2 -19553.819} C_VEL
LIN {X 0,Y 244.025,Z 348.81,A -85,B 0,C 180,E1 -19554.456,E2 -19554.456} C_VEL
LIN {X 0,Y 243.588,Z 336.603,A -85,B 0,C 180,E1 -19556.553,E2 -19556.553} C_VEL
LIN {X 0,Y 242.264,Z 325.887,A -85,B 0,C 180,E1 -19558.142,E2 -19558.142} C_VEL
LIN {X 0,Y 240.28,Z 315.539,A -85,B 0,C 180,E1 -19559.509,E2 -19559.509} C_VEL
LIN {X 0,Y 237.582,Z 305.152,A -85,B 0,C 180,E1 -19560.745,E2 -19560.745} C_VEL
LIN {X 0,Y 234.581,Z 295.766,A -85,B 0,C 180,E1 -19561.761,E2 -19561.761} C_VEL
LIN {X 0,Y 234.44,Z 294.813,A -85,B 0,C 180,E1 -19561.855,E2 -19561.855} C_VEL
LIN {X 0,Y 235.166,Z 291.436,A -85,B 0,C 180,E1 -19566.194,E2 -19566.194} C_VEL
LIN {X 0,Y 235.696,Z 289.29,A -85,B 0,C 180,E1 -19569.159,E2 -19569.159} C_VEL
LIN {X 0,Y 236.017,Z 287.384,A -85,B 0,C 180,E1 -19571.878,E2 -19571.878} C_VEL
LIN {X 0,Y 236.05,Z 284.948,A -85,B 0,C 180,E1 -19575.606,E2 -19575.606} C_VEL
LIN {X 0,Y 235.84,Z 282.907,A -85,B 0,C 180,E1 -19579.025,E2 -19579.025} C_VEL
LIN {X 0,Y 235.416,Z 280.376,A -85,B 0,C 180,E1 -19583.71,E2 -19583.71} C_VEL
LIN {X 0,Y 235.179,Z 278.549,A -85,B 0,C 180,E1 -19587.449,E2 -19587.449} C_VEL
LIN {X 0,Y 234.907,Z 276.834,A -85,B 0,C 180,E1 -19591.391,E2 -19591.391} C_VEL
LIN {X 0,Y 234.909,Z 276.729,A -85,B 0,C 180,E1 -19595.229,E2 -19595.229} C_VEL
LIN {X 0,Y 234.944,Z 276.723,A -85,B 0,C 180,E1 -19598.954,E2 -19598.954} C_VEL
LIN {X 0,Y 235.056,Z 276.705,A -85,B 0,C 180,E1 -19603.089,E2 -19603.089} C_VEL
LIN {X 0,Y 235.087,Z 276.703,A -85,B 0,C 180,E1 -19607.911,E2 -19607.911} C_VEL
LIN {X 0,Y 235.316,Z 276.673,A -85,B 0,C 180,E1 -19611.402,E2 -19611.402} C_VEL
LIN {X 0,Y 235.351,Z 276.667,A -85,B 0,C 180,E1 -19613.13,E2 -19613.13} C_VEL
LIN {X 0,Y 235.574,Z 276.637,A -85,B 0,C 180,E1 -19618.281,E2 -19618.281} C_VEL
LIN {X 0,Y 235.573,Z 276.618,A -85,B 0,C 180,E1 -19621.7,E2 -19621.7} C_VEL
LIN {X 0,Y 235.35,Z 276.668,A -85,B 0,C 180,E1 -19626.85,E2 -19626.85} C_VEL
LIN {X 0,Y 235.2,Z 276.682,A -85,B 0,C 180,E1 -19630.317,E2 -19630.317} C_VEL
LIN {X 0,Y 235.063,Z 276.702,A -85,B 0,C 180,E1 -19635.599,E2 -19635.599} C_VEL
LIN {X 0,Y 234.968,Z 276.712,A -85,B 0,C 180,E1 -19639.197,E2 -19639.197} C_VEL
LIN {X 0,Y 234.93,Z 276.723,A -85,B 0,C 180,E1 -19642.874,E2 -19642.874} C_VEL
LIN {X 0,Y 234.945,Z 276.718,A -85,B 0,C 180,E1 -19646.647,E2 -19646.647} C_VEL
LIN {X 0,Y 234.904,Z 276.726,A -85,B 0,C 180,E1 -19650.558,E2 -19650.558} C_VEL
LIN {X 0,Y 234.93,Z 276.723,A -85,B 0,C 180,E1 -19654.624,E2 -19654.624} C_VEL
LIN {X 0,Y 234.933,Z 276.721,A -85,B 0,C 180,E1 -19658.943,E2 -19658.943} C_VEL
LIN {X 0,Y 234.949,Z 276.718,A -85,B 0,C 180,E1 -19663.455,E2 -19663.455} C_VEL
LIN {X 0,Y 234.947,Z 276.719,A -85,B 0,C 180,E1 -19666.529,E2 -19666.529} C_VEL
LIN {X 0,Y 234.913,Z 276.723,A -85,B 0,C 180,E1 -19671.079,E2 -19671.079} C_VEL
LIN {X 0,Y 234.889,Z 276.726,A -85,B 0,C 180,E1 -19675.356,E2 -19675.356} C_VEL
LIN {X 0,Y 234.907,Z 276.799,A -85,B 0,C 180,E1 -19677.963,E2 -19677.963} C_VEL
LIN {X 0,Y 235.833,Z 279.498,A -85,B 0,C 180,E1 -19678.222,E2 -19678.222} C_VEL
LIN {X 0,Y 237.687,Z 282.781,A -85,B 0,C 180,E1 -19678.655,E2 -19678.655} C_VEL
LIN {X 0,Y 242.897,Z 292.981,A -85,B 0,C 180,E1 -19680.001,E2 -19680.001} C_VEL
LIN {X 0,Y 247.651,Z 304.398,A -85,B 0,C 180,E1 -19681.585,E2 -19681.585} C_VEL
LIN {X 0,Y 251.847,Z 314.727,A -85,B 0,C 180,E1 -19683.223,E2 -19683.223} C_VEL
LIN {X 0,Y 257.304,Z 324.703,A -85,B 0,C 180,E1 -19685.17,E2 -19685.17} C_VEL
LIN {X 0,Y 263.122,Z 333.167,A -85,B 0,C 180,E1 -19687.115,E2 -19687.115} C_VEL
LIN {X 0,Y 270.334,Z 341.846,A -85,B 0,C 180,E1 -19689.341,E2 -19689.341} C_VEL
LIN {X 0,Y 279.38,Z 351.033,A -85,B 0,C 180,E1 -19692.014,E2 -19692.014} C_VEL
LIN {X 0,Y 288.329,Z 359.102,A -85,B 0,C 180,E1 -19694.636,E2 -19694.636} C_VEL
LIN {X 0,Y 295.755,Z 365.417,A -85,B 0,C 180,E1 -19696.927,E2 -19696.927} C_VEL
LIN {X 0,Y 300.992,Z 369.684,A -85,B 0,C 180,E1 -19698.661,E2 -19698.661} C_VEL
LIN {X 0,Y 306.552,Z 374.244,A -85,B 0,C 180,E1 -19700.765,E2 -19700.765} C_VEL
LIN {X 0,Y 309.698,Z 376.835,A -85,B 0,C 180,E1 -19702.175,E2 -19702.175} C_VEL
LIN {X 0,Y 312.001,Z 378.878,A -85,B 0,C 180,E1 -19703.533,E2 -19703.533} C_VEL
LIN {X 0,Y 313.962,Z 380.529,A -85,B 0,C 180,E1 -19704.863,E2 -19704.863} C_VEL
LIN {X 0,Y 316.683,Z 382.169,A -85,B 0,C 180,E1 -19706.835,E2 -19706.835} C_VEL
LIN {X 0,Y 318.477,Z 382.848,A -85,B 0,C 180,E1 -19708.736,E2 -19708.736} C_VEL
LIN {X 0,Y 319.042,Z 382.952,A -85,B 0,C 180,E1 -19710,E2 -19710} C_VEL
LIN {X 0,Y 318.477,Z 382.844,A -85,B 0,C 180,E1 -19711.264,E2 -19711.264} C_VEL
LIN {X 0,Y 316.677,Z 382.176,A -85,B 0,C 180,E1 -19713.145,E2 -19713.145} C_VEL
LIN {X 0,Y 313.965,Z 380.514,A -85,B 0,C 180,E1 -19715.137,E2 -19715.137} C_VEL
LIN {X 0,Y 311.391,Z 378.349,A -85,B 0,C 180,E1 -19716.844,E2 -19716.844} C_VEL
LIN {X 0,Y 308.303,Z 375.611,A -85,B 0,C 180,E1 -19718.521,E2 -19718.521} C_VEL
LIN {X 0,Y 302.73,Z 371.144,A -85,B 0,C 180,E1 -19720.703,E2 -19720.703} C_VEL
LIN {X 0,Y 296.601,Z 366.105,A -85,B 0,C 180,E1 -19722.8,E2 -19722.8} C_VEL
LIN {X 0,Y 290.555,Z 361.038,A -85,B 0,C 180,E1 -19724.686,E2 -19724.686} C_VEL
LIN {X 0,Y 281.22,Z 352.756,A -85,B 0,C 180,E1 -19727.451,E2 -19727.451} C_VEL
LIN {X 0,Y 272.135,Z 343.725,A -85,B 0,C 180,E1 -19730.13,E2 -19730.13} C_VEL
LIN {X 0,Y 264.467,Z 334.853,A -85,B 0,C 180,E1 -19732.472,E2 -19732.472} C_VEL
LIN {X 0,Y 258.354,Z 326.408,A -85,B 0,C 180,E1 -19734.46,E2 -19734.46} C_VEL
LIN {X 0,Y 252.441,Z 315.971,A -85,B 0,C 180,E1 -19736.557,E2 -19736.557} C_VEL
LIN {X 0,Y 248.056,Z 305.54,A -85,B 0,C 180,E1 -19738.258,E2 -19738.258} C_VEL
LIN {X 0,Y 243.095,Z 293.37,A -85,B 0,C 180,E1 -19739.945,E2 -19739.945} C_VEL
LIN {X 0,Y 237.023,Z 281.402,A -85,B 0,C 180,E1 -19741.526,E2 -19741.526} C_VEL
LIN {X 0,Y 235.154,Z 277.915,A -85,B 0,C 180,E1 -19741.957,E2 -19741.957} C_VEL
LIN {X 0,Y 234.895,Z 276.727,A -85,B 0,C 180,E1 -19742.086,E2 -19742.086} C_VEL
LIN {X 0,Y 234.891,Z 276.725,A -85,B 0,C 180,E1 -19746.755,E2 -19746.755} C_VEL
LIN {X 0,Y 234.909,Z 276.723,A -85,B 0,C 180,E1 -19751.161,E2 -19751.161} C_VEL
LIN {X 0,Y 234.927,Z 276.721,A -85,B 0,C 180,E1 -19754.13,E2 -19754.13} C_VEL
LIN {X 0,Y 234.931,Z 276.72,A -85,B 0,C 180,E1 -19758.406,E2 -19758.406} C_VEL
LIN {X 0,Y 234.921,Z 276.723,A -85,B 0,C 180,E1 -19761.095,E2 -19761.095} C_VEL
LIN {X 0,Y 234.93,Z 276.723,A -85,B 0,C 180,E1 -19765.376,E2 -19765.376} C_VEL
LIN {X 0,Y 234.942,Z 276.719,A -85,B 0,C 180,E1 -19770.167,E2 -19770.167} C_VEL
LIN {X 0,Y 234.97,Z 276.713,A -85,B 0,C 180,E1 -19773.804,E2 -19773.804} C_VEL
LIN {X 0,Y 234.969,Z 276.713,A -85,B 0,C 180,E1 -19778.978,E2 -19778.978} C_VEL
LIN {X 0,Y 235.039,Z 276.707,A -85,B 0,C 180,E1 -19783.102,E2 -19783.102} C_VEL
LIN {X 0,Y 235.085,Z 276.701,A -85,B 0,C 180,E1 -19787.931,E2 -19787.931} C_VEL
LIN {X 0,Y 235.312,Z 276.671,A -85,B 0,C 180,E1 -19791.422,E2 -19791.422} C_VEL
LIN {X 0,Y 235.35,Z 276.668,A -85,B 0,C 180,E1 -19793.15,E2 -19793.15} C_VEL
LIN {X 0,Y 235.573,Z 276.618,A -85,B 0,C 180,E1 -19798.3,E2 -19798.3} C_VEL
LIN {X 0,Y 235.574,Z 276.637,A -85,B 0,C 180,E1 -19801.719,E2 -19801.719} C_VEL
LIN {X 0,Y 235.351,Z 276.668,A -85,B 0,C 180,E1 -19806.87,E2 -19806.87} C_VEL
LIN {X 0,Y 235.186,Z 276.69,A -85,B 0,C 180,E1 -19810.338,E2 -19810.338} C_VEL
LIN {X 0,Y 235.062,Z 276.707,A -85,B 0,C 180,E1 -19815.619,E2 -19815.619} C_VEL
LIN {X 0,Y 234.966,Z 276.717,A -85,B 0,C 180,E1 -19819.219,E2 -19819.219} C_VEL
LIN {X 0,Y 234.917,Z 276.723,A -85,B 0,C 180,E1 -19822.897,E2 -19822.897} C_VEL
LIN {X 0,Y 234.933,Z 276.721,A -85,B 0,C 180,E1 -19826.671,E2 -19826.671} C_VEL
LIN {X 0,Y 234.907,Z 276.835,A -85,B 0,C 180,E1 -19828.609,E2 -19828.609} C_VEL
LIN {X 0,Y 235.24,Z 278.867,A -85,B 0,C 180,E1 -19833.227,E2 -19833.227} C_VEL
LIN {X 0,Y 235.444,Z 280.58,A -85,B 0,C 180,E1 -19836.665,E2 -19836.665} C_VEL
LIN {X 0,Y 235.829,Z 282.928,A -85,B 0,C 180,E1 -19840.977,E2 -19840.977} C_VEL
LIN {X 0,Y 236.112,Z 285.73,A -85,B 0,C 180,E1 -19845.602,E2 -19845.602} C_VEL
LIN {X 0,Y 235.92,Z 288.035,A -85,B 0,C 180,E1 -19849.053,E2 -19849.053} C_VEL
LIN {X 0,Y 235.639,Z 289.592,A -85,B 0,C 180,E1 -19851.221,E2 -19851.221} C_VEL
LIN {X 0,Y 234.896,Z 292.657,A -85,B 0,C 180,E1 -19855.357,E2 -19855.357} C_VEL
LIN {X 0,Y 234.439,Z 294.803,A -85,B 0,C 180,E1 -19858.144,E2 -19858.144} C_VEL
LIN {X 0,Y 235.436,Z 298.329,A -85,B 0,C 180,E1 -19858.487,E2 -19858.487} C_VEL
LIN {X 0,Y 239.006,Z 310.262,A -85,B 0,C 180,E1 -19859.827,E2 -19859.827} C_VEL
LIN {X 0,Y 241.356,Z 320.781,A -85,B 0,C 180,E1 -19861.148,E2 -19861.148} C_VEL
LIN {X 0,Y 241.591,Z 326.155,A -85,B 0,C 180,E1 -19861.795,E2 -19861.795} C_VEL
LIN {X 0,Y 239.982,Z 334.913,A -85,B 0,C 180,E1 -19862.784,E2 -19862.784} C_VEL
LIN {X 0,Y 237.855,Z 343.514,A -85,B 0,C 180,E1 -19863.903,E2 -19863.903} C_VEL
LIN {X 0,Y 237.31,Z 348.315,A -85,B 0,C 180,E1 -19864.748,E2 -19864.748} C_VEL
LIN {X 0,Y 237.125,Z 352.014,A -85,B 0,C 180,E1 -19865.485,E2 -19865.485} C_VEL
LIN {X 0,Y 235.072,Z 360.193,A -85,B 0,C 180,E1 -19867.129,E2 -19867.129} C_VEL
LIN {X 0,Y 232.74,Z 369.478,A -85,B 0,C 180,E1 -19869.426,E2 -19869.426} C_VEL
LIN {X 0,Y 230.725,Z 377.083,A -85,B 0,C 180,E1 -19871.807,E2 -19871.807} C_VEL
LIN {X 0,Y 229.179,Z 382.744,A -85,B 0,C 180,E1 -19873.979,E2 -19873.979} C_VEL
LIN {X 0,Y 227.652,Z 388.238,A -85,B 0,C 180,E1 -19876.613,E2 -19876.613} C_VEL
LIN {X 0,Y 226.653,Z 392.57,A -85,B 0,C 180,E1 -19879.278,E2 -19879.278} C_VEL
LIN {X 0,Y 226.189,Z 394.941,A -85,B 0,C 180,E1 -19881.063,E2 -19881.063} C_VEL
LIN {X 0,Y 225.714,Z 398.138,A -85,B 0,C 180,E1 -19884.64,E2 -19884.64} C_VEL
LIN {X 0,Y 225.62,Z 399.201,A -85,B 0,C 180,E1 -19886.428,E2 -19886.428} C_VEL
LIN {X 0,Y 225.641,Z 399.795,A -85,B 0,C 180,E1 -19888.215,E2 -19888.215} C_VEL
LIN {X 0,Y 225.705,Z 399.952,A -85,B 0,C 180,E1 -19890,E2 -19890} C_VEL
LIN {X 0,Y 225.641,Z 399.795,A -85,B 0,C 180,E1 -19891.785,E2 -19891.785} C_VEL
LIN {X 0,Y 225.682,Z 398.577,A -85,B 0,C 180,E1 -19894.701,E2 -19894.701} C_VEL
LIN {X 0,Y 225.868,Z 396.745,A -85,B 0,C 180,E1 -19897.15,E2 -19897.15} C_VEL
LIN {X 0,Y 226.401,Z 393.789,A -85,B 0,C 180,E1 -19899.83,E2 -19899.83} C_VEL
LIN {X 0,Y 227.307,Z 389.795,A -85,B 0,C 180,E1 -19902.499,E2 -19902.499} C_VEL
LIN {X 0,Y 228.614,Z 384.66,A -85,B 0,C 180,E1 -19905.147,E2 -19905.147} C_VEL
LIN {X 0,Y 230.119,Z 379.397,A -85,B 0,C 180,E1 -19907.324,E2 -19907.324} C_VEL
LIN {X 0,Y 231.857,Z 373.078,A -85,B 0,C 180,E1 -19909.477,E2 -19909.477} C_VEL
LIN {X 0,Y 233.741,Z 365.493,A -85,B 0,C 180,E1 -19911.612,E2 -19911.612} C_VEL
LIN {X 0,Y 236.038,Z 356.353,A -85,B 0,C 180,E1 -19913.7,E2 -19913.7} C_VEL
LIN {X 0,Y 237.289,Z 350.876,A -85,B 0,C 180,E1 -19914.73,E2 -19914.73} C_VEL
LIN {X 0,Y 237.189,Z 343.442,A -85,B 0,C 180,E1 -19916.151,E2 -19916.151} C_VEL
LIN {X 0,Y 236.81,Z 335.64,A -85,B 0,C 180,E1 -19917.483,E2 -19917.483} C_VEL
LIN {X 0,Y 235.494,Z 325.658,A -85,B 0,C 180,E1 -19919.027,E2 -19919.027} C_VEL
LIN {X 0,Y 233.726,Z 316.346,A -85,B 0,C 180,E1 -19920.323,E2 -19920.323} C_VEL
LIN {X 0,Y 230.896,Z 305.576,A -85,B 0,C 180,E1 -19921.689,E2 -19921.689} C_VEL
LIN {X 0,Y 228.208,Z 297.379,A -85,B 0,C 180,E1 -19922.666,E2 -19922.666} C_VEL
LIN {X 0,Y 227.556,Z 294.624,A -85,B 0,C 180,E1 -19922.914,E2 -19922.914} C_VEL
LIN {X 0,Y 228.396,Z 290.886,A -85,B 0,C 180,E1 -19927.982,E2 -19927.982} C_VEL
LIN {X 0,Y 228.753,Z 289.366,A -85,B 0,C 180,E1 -19930.179,E2 -19930.179} C_VEL
LIN {X 0,Y 228.979,Z 287.786,A -85,B 0,C 180,E1 -19932.544,E2 -19932.544} C_VEL
LIN {X 0,Y 229.013,Z 286.158,A -85,B 0,C 180,E1 -19935.093,E2 -19935.093} C_VEL
LIN {X 0,Y 228.899,Z 284.741,A -85,B 0,C 180,E1 -19937.498,E2 -19937.498} C_VEL
LIN {X 0,Y 228.665,Z 283.235,A -85,B 0,C 180,E1 -19940.207,E2 -19940.207} C_VEL
LIN {X 0,Y 228.359,Z 281.165,A -85,B 0,C 180,E1 -19944.205,E2 -19944.205} C_VEL
LIN {X 0,Y 228.059,Z 279.213,A -85,B 0,C 180,E1 -19948.397,E2 -19948.397} C_VEL
LIN {X 0,Y 227.846,Z 277.607,A -85,B 0,C 180,E1 -19952.43,E2 -19952.43} C_VEL
LIN {X 0,Y 227.865,Z 277.608,A -85,B 0,C 180,E1 -19956.352,E2 -19956.352} C_VEL
LIN {X 0,Y 227.895,Z 277.602,A -85,B 0,C 180,E1 -19960.161,E2 -19960.161} C_VEL
LIN {X 0,Y 228.014,Z 277.584,A -85,B 0,C 180,E1 -19963.885,E2 -19963.885} C_VEL
LIN {X 0,Y 228.127,Z 277.568,A -85,B 0,C 180,E1 -19969.338,E2 -19969.338} C_VEL
LIN {X 0,Y 228.303,Z 277.545,A -85,B 0,C 180,E1 -19972.917,E2 -19972.917} C_VEL
LIN {X 0,Y 228.532,Z 277.514,A -85,B 0,C 180,E1 -19978.228,E2 -19978.228} C_VEL
LIN {X 0,Y 228.531,Z 277.493,A -85,B 0,C 180,E1 -19981.752,E2 -19981.752} C_VEL
LIN {X 0,Y 228.302,Z 277.546,A -85,B 0,C 180,E1 -19987.062,E2 -19987.062} C_VEL
LIN {X 0,Y 228.13,Z 277.563,A -85,B 0,C 180,E1 -19990.641,E2 -19990.641} C_VEL
LIN {X 0,Y 228.022,Z 277.577,A -85,B 0,C 180,E1 -19994.263,E2 -19994.263} C_VEL
LIN {X 0,Y 227.935,Z 277.591,A -85,B 0,C 180,E1 -19997.947,E2 -19997.947} C_VEL
LIN {X 0,Y 227.894,Z 277.597,A -85,B 0,C 180,E1 -20002.309,E2 -20002.309} C_VEL
LIN {X 0,Y 227.918,Z 277.593,A -85,B 0,C 180,E1 -20006.592,E2 -20006.592} C_VEL
LIN {X 0,Y 227.881,Z 277.599,A -85,B 0,C 180,E1 -20010.286,E2 -20010.286} C_VEL
LIN {X 0,Y 227.859,Z 277.6,A -85,B 0,C 180,E1 -20013.709,E2 -20013.709} C_VEL
LIN {X 0,Y 227.838,Z 277.604,A -85,B 0,C 180,E1 -20018.076,E2 -20018.076} C_VEL
LIN {X 0,Y 227.885,Z 277.598,A -85,B 0,C 180,E1 -20022.708,E2 -20022.708} C_VEL
LIN {X 0,Y 227.882,Z 277.597,A -85,B 0,C 180,E1 -20027.275,E2 -20027.275} C_VEL
LIN {X 0,Y 227.825,Z 277.608,A -85,B 0,C 180,E1 -20031.906,E2 -20031.906} C_VEL
LIN {X 0,Y 227.835,Z 277.606,A -85,B 0,C 180,E1 -20036.37,E2 -20036.37} C_VEL
LIN {X 0,Y 227.859,Z 277.602,A -85,B 0,C 180,E1 -20036.842,E2 -20036.842} C_VEL
LIN {X 0,Y 228.977,Z 280.636,A -85,B 0,C 180,E1 -20037.197,E2 -20037.197} C_VEL
LIN {X 0,Y 230.282,Z 282.932,A -85,B 0,C 180,E1 -20037.521,E2 -20037.521} C_VEL
LIN {X 0,Y 235.094,Z 292.091,A -85,B 0,C 180,E1 -20038.815,E2 -20038.815} C_VEL
LIN {X 0,Y 239.503,Z 302.032,A -85,B 0,C 180,E1 -20040.274,E2 -20040.274} C_VEL
LIN {X 0,Y 243.893,Z 313.805,A -85,B 0,C 180,E1 -20042.133,E2 -20042.133} C_VEL
LIN {X 0,Y 248.004,Z 322.725,A -85,B 0,C 180,E1 -20043.838,E2 -20043.838} C_VEL
LIN {X 0,Y 252.672,Z 330.617,A -85,B 0,C 180,E1 -20045.604,E2 -20045.604} C_VEL
LIN {X 0,Y 259.55,Z 339.969,A -85,B 0,C 180,E1 -20047.999,E2 -20047.999} C_VEL
LIN {X 0,Y 268.007,Z 349.207,A -85,B 0,C 180,E1 -20050.704,E2 -20050.704} C_VEL
LIN {X 0,Y 276.791,Z 357.48,A -85,B 0,C 180,E1 -20053.436,E2 -20053.436} C_VEL
LIN {X 0,Y 284.171,Z 363.568,A -85,B 0,C 180,E1 -20055.682,E2 -20055.682} C_VEL
LIN {X 0,Y 289.506,Z 367.804,A -85,B 0,C 180,E1 -20057.38,E2 -20057.38} C_VEL
LIN {X 0,Y 294.251,Z 371.403,A -85,B 0,C 180,E1 -20058.985,E2 -20058.985} C_VEL
LIN {X 0,Y 300.465,Z 376.106,A -85,B 0,C 180,E1 -20061.387,E2 -20061.387} C_VEL
LIN {X 0,Y 303.227,Z 378.24,A -85,B 0,C 180,E1 -20062.677,E2 -20062.677} C_VEL
LIN {X 0,Y 306.502,Z 381.02,A -85,B 0,C 180,E1 -20064.738,E2 -20064.738} C_VEL
LIN {X 0,Y 309.605,Z 382.945,A -85,B 0,C 180,E1 -20066.97,E2 -20066.97} C_VEL
LIN {X 0,Y 311.312,Z 383.678,A -85,B 0,C 180,E1 -20068.706,E2 -20068.706} C_VEL
LIN {X 0,Y 311.969,Z 383.83,A -85,B 0,C 180,E1 -20070,E2 -20070} C_VEL
LIN {X 0,Y 311.311,Z 383.677,A -85,B 0,C 180,E1 -20071.294,E2 -20071.294} C_VEL
LIN {X 0,Y 309.6,Z 382.955,A -85,B 0,C 180,E1 -20073.014,E2 -20073.014} C_VEL
LIN {X 0,Y 306.503,Z 381.02,A -85,B 0,C 180,E1 -20075.262,E2 -20075.262} C_VEL
LIN {X 0,Y 303.225,Z 378.24,A -85,B 0,C 180,E1 -20077.323,E2 -20077.323} C_VEL
LIN {X 0,Y 300.467,Z 376.109,A -85,B 0,C 180,E1 -20078.612,E2 -20078.612} C_VEL
LIN {X 0,Y 294.231,Z 371.404,A -85,B 0,C 180,E1 -20081.016,E2 -20081.016} C_VEL
LIN {X 0,Y 287.12,Z 365.898,A -85,B 0,C 180,E1 -20083.401,E2 -20083.401} C_VEL
LIN {X 0,Y 280.605,Z 360.689,A -85,B 0,C 180,E1 -20085.41,E2 -20085.41} C_VEL
LIN {X 0,Y 271.892,Z 353.04,A -85,B 0,C 180,E1 -20088.07,E2 -20088.07} C_VEL
LIN {X 0,Y 263.133,Z 344.076,A -85,B 0,C 180,E1 -20090.836,E2 -20090.836} C_VEL
LIN {X 0,Y 255.797,Z 335.171,A -85,B 0,C 180,E1 -20093.273,E2 -20093.273} C_VEL
LIN {X 0,Y 250.378,Z 326.954,A -85,B 0,C 180,E1 -20095.248,E2 -20095.248} C_VEL
LIN {X 0,Y 245.315,Z 317.031,A -85,B 0,C 180,E1 -20097.282,E2 -20097.282} C_VEL
LIN {X 0,Y 241.183,Z 306.391,A -85,B 0,C 180,E1 -20099.077,E2 -20099.077} C_VEL
LIN {X 0,Y 236.564,Z 295.222,A -85,B 0,C 180,E1 -20100.743,E2 -20100.743} C_VEL
LIN {X 0,Y 231.211,Z 284.519,A -85,B 0,C 180,E1 -20102.271,E2 -20102.271} C_VEL
LIN {X 0,Y 228.063,Z 278.605,A -85,B 0,C 180,E1 -20103.055,E2 -20103.055} C_VEL
LIN {X 0,Y 227.855,Z 277.603,A -85,B 0,C 180,E1 -20103.157,E2 -20103.157} C_VEL
LIN {X 0,Y 227.853,Z 277.602,A -85,B 0,C 180,E1 -20106.705,E2 -20106.705} C_VEL
LIN {X 0,Y 227.854,Z 277.601,A -85,B 0,C 180,E1 -20110.37,E2 -20110.37} C_VEL
LIN {X 0,Y 227.878,Z 277.598,A -85,B 0,C 180,E1 -20114.836,E2 -20114.836} C_VEL
LIN {X 0,Y 227.882,Z 277.6,A -85,B 0,C 180,E1 -20117.745,E2 -20117.745} C_VEL
LIN {X 0,Y 227.838,Z 277.604,A -85,B 0,C 180,E1 -20121.924,E2 -20121.924} C_VEL
LIN {X 0,Y 227.86,Z 277.599,A -85,B 0,C 180,E1 -20126.383,E2 -20126.383} C_VEL
LIN {X 0,Y 227.892,Z 277.597,A -85,B 0,C 180,E1 -20130.448,E2 -20130.448} C_VEL
LIN {X 0,Y 227.901,Z 277.593,A -85,B 0,C 180,E1 -20134.436,E2 -20134.436} C_VEL
LIN {X 0,Y 227.923,Z 277.593,A -85,B 0,C 180,E1 -20138.296,E2 -20138.296} C_VEL
LIN {X 0,Y 228.007,Z 277.581,A -85,B 0,C 180,E1 -20143.906,E2 -20143.906} C_VEL
LIN {X 0,Y 228.042,Z 277.578,A -85,B 0,C 180,E1 -20147.553,E2 -20147.553} C_VEL
LIN {X 0,Y 228.25,Z 277.551,A -85,B 0,C 180,E1 -20151.155,E2 -20151.155} C_VEL
LIN {X 0,Y 228.302,Z 277.546,A -85,B 0,C 180,E1 -20152.938,E2 -20152.938} C_VEL
LIN {X 0,Y 228.531,Z 277.493,A -85,B 0,C 180,E1 -20158.248,E2 -20158.248} C_VEL
LIN {X 0,Y 228.532,Z 277.514,A -85,B 0,C 180,E1 -20161.772,E2 -20161.772} C_VEL
LIN {X 0,Y 228.303,Z 277.546,A -85,B 0,C 180,E1 -20167.083,E2 -20167.083} C_VEL
LIN {X 0,Y 228.127,Z 277.568,A -85,B 0,C 180,E1 -20170.662,E2 -20170.662} C_VEL
LIN {X 0,Y 228.014,Z 277.584,A -85,B 0,C 180,E1 -20176.115,E2 -20176.115} C_VEL
LIN {X 0,Y 227.927,Z 277.595,A -85,B 0,C 180,E1 -20181.726,E2 -20181.726} C_VEL
LIN {X 0,Y 227.912,Z 277.595,A -85,B 0,C 180,E1 -20186.589,E2 -20186.589} C_VEL
LIN {X 0,Y 227.854,Z 277.603,A -85,B 0,C 180,E1 -20187.569,E2 -20187.569} C_VEL
LIN {X 0,Y 228.069,Z 279.215,A -85,B 0,C 180,E1 -20191.601,E2 -20191.601} C_VEL
LIN {X 0,Y 228.365,Z 281.166,A -85,B 0,C 180,E1 -20195.794,E2 -20195.794} C_VEL
LIN {X 0,Y 228.699,Z 283.459,A -85,B 0,C 180,E1 -20200.201,E2 -20200.201} C_VEL
LIN {X 0,Y 228.894,Z 284.785,A -85,B 0,C 180,E1 -20202.533,E2 -20202.533} C_VEL
LIN {X 0,Y 229.031,Z 286.325,A -85,B 0,C 180,E1 -20205.109,E2 -20205.109} C_VEL
LIN {X 0,Y 228.98,Z 287.85,A -85,B 0,C 180,E1 -20207.528,E2 -20207.528} C_VEL
LIN {X 0,Y 228.703,Z 289.639,A -85,B 0,C 180,E1 -20210.208,E2 -20210.208} C_VEL
LIN {X 0,Y 228.003,Z 292.441,A -85,B 0,C 180,E1 -20214.151,E2 -20214.151} C_VEL
LIN {X 0,Y 227.523,Z 294.615,A -85,B 0,C 180,E1 -20217.087,E2 -20217.087} C_VEL
LIN {X 0,Y 228.354,Z 297.736,A -85,B 0,C 180,E1 -20217.374,E2 -20217.374} C_VEL
LIN {X 0,Y 232.412,Z 310.804,A -85,B 0,C 180,E1 -20218.952,E2 -20218.952} C_VEL
LIN {X 0,Y 234.893,Z 322.15,A -85,B 0,C 180,E1 -20220.468,E2 -20220.468} C_VEL
LIN {X 0,Y 236.28,Z 331.187,A -85,B 0,C 180,E1 -20221.8,E2 -20221.8} C_VEL
LIN {X 0,Y 237.103,Z 339.805,A -85,B 0,C 180,E1 -20223.205,E2 -20223.205} C_VEL
LIN {X 0,Y 237.31,Z 348.315,A -85,B 0,C 180,E1 -20224.748,E2 -20224.748} C_VEL
LIN {X 0,Y 236.694,Z 350.911,A -85,B 0,C 180,E1 -20225.212,E2 -20225.212} C_VEL
LIN {X 0,Y 234.485,Z 354.529,A -85,B 0,C 180,E1 -20225.728,E2 -20225.728} C_VEL
LIN {X 0,Y 228.912,Z 361.125,A -85,B 0,C 180,E1 -20226.733,E2 -20226.733} C_VEL
LIN {X 0,Y 227.486,Z 363.942,A -85,B 0,C 180,E1 -20227.369,E2 -20227.369} C_VEL
LIN {X 0,Y 225.646,Z 371.095,A -85,B 0,C 180,E1 -20229.353,E2 -20229.353} C_VEL
LIN {X 0,Y 223.603,Z 378.027,A -85,B 0,C 180,E1 -20231.681,E2 -20231.681} C_VEL
LIN {X 0,Y 222.343,Z 382.532,A -85,B 0,C 180,E1 -20233.473,E2 -20233.473} C_VEL
LIN {X 0,Y 220.71,Z 388.025,A -85,B 0,C 180,E1 -20236.183,E2 -20236.183} C_VEL
LIN {X 0,Y 219.661,Z 392.358,A -85,B 0,C 180,E1 -20238.933,E2 -20238.933} C_VEL
LIN {X 0,Y 219.141,Z 394.729,A -85,B 0,C 180,E1 -20240.773,E2 -20240.773} C_VEL
LIN {X 0,Y 218.792,Z 396.533,A -85,B 0,C 180,E1 -20242.618,E2 -20242.618} C_VEL
LIN {X 0,Y 218.525,Z 398.989,A -85,B 0,C 180,E1 -20246.312,E2 -20246.312} C_VEL
LIN {X 0,Y 218.542,Z 399.583,A -85,B 0,C 180,E1 -20248.157,E2 -20248.157} C_VEL
LIN {X 0,Y 218.622,Z 399.741,A -85,B 0,C 180,E1 -20250,E2 -20250} C_VEL
LIN {X 0,Y 218.542,Z 399.583,A -85,B 0,C 180,E1 -20251.843,E2 -20251.843} C_VEL
LIN {X 0,Y 218.575,Z 398.581,A -85,B 0,C 180,E1 -20254.518,E2 -20254.518} C_VEL
LIN {X 0,Y 218.82,Z 396.534,A -85,B 0,C 180,E1 -20257.381,E2 -20257.381} C_VEL
LIN {X 0,Y 219.383,Z 393.577,A -85,B 0,C 180,E1 -20260.148,E2 -20260.148} C_VEL
LIN {X 0,Y 220.326,Z 389.582,A -85,B 0,C 180,E1 -20262.902,E2 -20262.902} C_VEL
LIN {X 0,Y 221.748,Z 384.448,A -85,B 0,C 180,E1 -20265.628,E2 -20265.628} C_VEL
LIN {X 0,Y 223.296,Z 379.184,A -85,B 0,C 180,E1 -20267.87,E2 -20267.87} C_VEL
LIN {X 0,Y 225.145,Z 372.866,A -85,B 0,C 180,E1 -20270.082,E2 -20270.082} C_VEL
LIN {X 0,Y 226.693,Z 366.909,A -85,B 0,C 180,E1 -20271.84,E2 -20271.84} C_VEL
LIN {X 0,Y 228.499,Z 359.98,A -85,B 0,C 180,E1 -20273.568,E2 -20273.568} C_VEL
LIN {X 0,Y 230.576,Z 351.799,A -85,B 0,C 180,E1 -20275.259,E2 -20275.259} C_VEL
LIN {X 0,Y 230.551,Z 344.583,A -85,B 0,C 180,E1 -20276.719,E2 -20276.719} C_VEL
LIN {X 0,Y 230.145,Z 336.079,A -85,B 0,C 180,E1 -20278.249,E2 -20278.249} C_VEL
LIN {X 0,Y 228.756,Z 325.427,A -85,B 0,C 180,E1 -20279.968,E2 -20279.968} C_VEL
LIN {X 0,Y 227.12,Z 316.679,A -85,B 0,C 180,E1 -20281.246,E2 -20281.246} C_VEL
LIN {X 0,Y 224.101,Z 305.355,A -85,B 0,C 180,E1 -20282.767,E2 -20282.767} C_VEL
LIN {X 0,Y 221.417,Z 297.428,A -85,B 0,C 180,E1 -20283.785,E2 -20283.785} C_VEL
LIN {X 0,Y 220.627,Z 294.389,A -85,B 0,C 180,E1 -20284.118,E2 -20284.118} C_VEL
LIN {X 0,Y 221.219,Z 292.03,A -85,B 0,C 180,E1 -20287.404,E2 -20287.404} C_VEL
LIN {X 0,Y 221.716,Z 289.96,A -85,B 0,C 180,E1 -20290.457,E2 -20290.457} C_VEL
LIN {X 0,Y 221.918,Z 287.622,A -85,B 0,C 180,E1 -20294.164,E2 -20294.164} C_VEL
LIN {X 0,Y 221.763,Z 285.252,A -85,B 0,C 180,E1 -20298.267,E2 -20298.267} C_VEL
LIN {X 0,Y 221.394,Z 282.836,A -85,B 0,C 180,E1 -20302.894,E2 -20302.894} C_VEL
LIN {X 0,Y 221.099,Z 280.785,A -85,B 0,C 180,E1 -20307.281,E2 -20307.281} C_VEL
LIN {X 0,Y 220.863,Z 279.038,A -85,B 0,C 180,E1 -20311.48,E2 -20311.48} C_VEL
LIN {X 0,Y 220.84,Z 278.48,A -85,B 0,C 180,E1 -20313.532,E2 -20313.532} C_VEL
LIN {X 0,Y 220.864,Z 278.479,A -85,B 0,C 180,E1 -20317.542,E2 -20317.542} C_VEL
LIN {X 0,Y 220.922,Z 278.467,A -85,B 0,C 180,E1 -20322.62,E2 -20322.62} C_VEL
LIN {X 0,Y 220.978,Z 278.458,A -85,B 0,C 180,E1 -20327.126,E2 -20327.126} C_VEL
LIN {X 0,Y 221.196,Z 278.431,A -85,B 0,C 180,E1 -20330.849,E2 -20330.849} C_VEL
LIN {X 0,Y 221.241,Z 278.425,A -85,B 0,C 180,E1 -20332.69,E2 -20332.69} C_VEL
LIN {X 0,Y 221.465,Z 278.395,A -85,B 0,C 180,E1 -20338.171,E2 -20338.171} C_VEL
LIN {X 0,Y 221.465,Z 278.372,A -85,B 0,C 180,E1 -20341.808,E2 -20341.808} C_VEL
LIN {X 0,Y 221.239,Z 278.428,A -85,B 0,C 180,E1 -20347.289,E2 -20347.289} C_VEL
LIN {X 0,Y 221.05,Z 278.446,A -85,B 0,C 180,E1 -20350.986,E2 -20350.986} C_VEL
LIN {X 0,Y 220.962,Z 278.459,A -85,B 0,C 180,E1 -20356.622,E2 -20356.622} C_VEL
LIN {X 0,Y 220.855,Z 278.467,A -85,B 0,C 180,E1 -20360.477,E2 -20360.477} C_VEL
LIN {X 0,Y 220.839,Z 278.472,A -85,B 0,C 180,E1 -20364.425,E2 -20364.425} C_VEL
LIN {X 0,Y 220.81,Z 278.48,A -85,B 0,C 180,E1 -20368.503,E2 -20368.503} C_VEL
LIN {X 0,Y 220.795,Z 278.483,A -85,B 0,C 180,E1 -20372.745,E2 -20372.745} C_VEL
LIN {X 0,Y 220.807,Z 278.48,A -85,B 0,C 180,E1 -20377.278,E2 -20377.278} C_VEL
LIN {X 0,Y 220.824,Z 278.479,A -85,B 0,C 180,E1 -20381.922,E2 -20381.922} C_VEL
LIN {X 0,Y 220.831,Z 278.476,A -85,B 0,C 180,E1 -20385.562,E2 -20385.562} C_VEL
LIN {X 0,Y 220.816,Z 278.48,A -85,B 0,C 180,E1 -20390.466,E2 -20390.466} C_VEL
LIN {X 0,Y 220.759,Z 278.487,A -85,B 0,C 180,E1 -20395.038,E2 -20395.038} C_VEL
LIN {X 0,Y 220.759,Z 278.487,A -85,B 0,C 180,E1 -20395.682,E2 -20395.682} C_VEL
LIN {X 0,Y 221.809,Z 281.388,A -85,B 0,C 180,E1 -20396.021,E2 -20396.021} C_VEL
LIN {X 0,Y 223.079,Z 283.307,A -85,B 0,C 180,E1 -20396.341,E2 -20396.341} C_VEL
LIN {X 0,Y 228.39,Z 293.526,A -85,B 0,C 180,E1 -20397.882,E2 -20397.882} C_VEL
LIN {X 0,Y 232.677,Z 303.011,A -85,B 0,C 180,E1 -20399.384,E2 -20399.384} C_VEL
LIN {X 0,Y 236.264,Z 312.733,A -85,B 0,C 180,E1 -20400.988,E2 -20400.988} C_VEL
LIN {X 0,Y 239.764,Z 321.782,A -85,B 0,C 180,E1 -20402.689,E2 -20402.689} C_VEL
LIN {X 0,Y 243.562,Z 329.299,A -85,B 0,C 180,E1 -20404.354,E2 -20404.354} C_VEL
LIN {X 0,Y 249.742,Z 338.838,A -85,B 0,C 180,E1 -20406.798,E2 -20406.798} C_VEL
LIN {X 0,Y 257.09,Z 347.613,A -85,B 0,C 180,E1 -20409.399,E2 -20409.399} C_VEL
LIN {X 0,Y 265.626,Z 356.09,A -85,B 0,C 180,E1 -20412.229,E2 -20412.229} C_VEL
LIN {X 0,Y 274.935,Z 363.85,A -85,B 0,C 180,E1 -20415.19,E2 -20415.19} C_VEL
LIN {X 0,Y 281.082,Z 368.457,A -85,B 0,C 180,E1 -20417.143,E2 -20417.143} C_VEL
LIN {X 0,Y 288.207,Z 373.568,A -85,B 0,C 180,E1 -20419.597,E2 -20419.597} C_VEL
LIN {X 0,Y 293.683,Z 377.369,A -85,B 0,C 180,E1 -20421.745,E2 -20421.745} C_VEL
LIN {X 0,Y 296.754,Z 379.516,A -85,B 0,C 180,E1 -20423.2,E2 -20423.2} C_VEL
LIN {X 0,Y 298.944,Z 381.247,A -85,B 0,C 180,E1 -20424.604,E2 -20424.604} C_VEL
LIN {X 0,Y 302.523,Z 383.384,A -85,B 0,C 180,E1 -20427.134,E2 -20427.134} C_VEL
LIN {X 0,Y 304.104,Z 384.064,A -85,B 0,C 180,E1 -20428.676,E2 -20428.676} C_VEL
LIN {X 0,Y 304.86,Z 384.246,A -85,B 0,C 180,E1 -20430,E2 -20430} C_VEL
LIN {X 0,Y 304.101,Z 384.064,A -85,B 0,C 180,E1 -20431.324,E2 -20431.324} C_VEL
LIN {X 0,Y 302.519,Z 383.392,A -85,B 0,C 180,E1 -20432.853,E2 -20432.853} C_VEL
LIN {X 0,Y 300.932,Z 382.571,A -85,B 0,C 180,E1 -20434.017,E2 -20434.017} C_VEL
LIN {X 0,Y 298.938,Z 381.247,A -85,B 0,C 180,E1 -20435.396,E2 -20435.396} C_VEL
LIN {X 0,Y 296.753,Z 379.516,A -85,B 0,C 180,E1 -20436.8,E2 -20436.8} C_VEL
LIN {X 0,Y 293.678,Z 377.369,A -85,B 0,C 180,E1 -20438.255,E2 -20438.255} C_VEL
LIN {X 0,Y 288.192,Z 373.566,A -85,B 0,C 180,E1 -20440.404,E2 -20440.404} C_VEL
LIN {X 0,Y 280.552,Z 368.078,A -85,B 0,C 180,E1 -20443.029,E2 -20443.029} C_VEL
LIN {X 0,Y 272.215,Z 361.731,A -85,B 0,C 180,E1 -20445.663,E2 -20445.663} C_VEL
LIN {X 0,Y 262.731,Z 353.319,A -85,B 0,C 180,E1 -20448.723,E2 -20448.723} C_VEL
LIN {X 0,Y 255.007,Z 345.347,A -85,B 0,C 180,E1 -20451.305,E2 -20451.305} C_VEL
LIN {X 0,Y 248.24,Z 336.774,A -85,B 0,C 180,E1 -20453.767,E2 -20453.767} C_VEL
LIN {X 0,Y 242.544,Z 327.37,A -85,B 0,C 180,E1 -20456.099,E2 -20456.099} C_VEL
LIN {X 0,Y 238.529,Z 318.808,A -85,B 0,C 180,E1 -20457.909,E2 -20457.909} C_VEL
LIN {X 0,Y 234.233,Z 306.989,A -85,B 0,C 180,E1 -20459.987,E2 -20459.987} C_VEL
LIN {X 0,Y 229.267,Z 295.293,A -85,B 0,C 180,E1 -20461.846,E2 -20461.846} C_VEL
LIN {X 0,Y 222.775,Z 282.566,A -85,B 0,C 180,E1 -20463.771,E2 -20463.771} C_VEL
LIN {X 0,Y 221.199,Z 280.122,A -85,B 0,C 180,E1 -20464.161,E2 -20464.161} C_VEL
LIN {X 0,Y 220.759,Z 278.487,A -85,B 0,C 180,E1 -20464.318,E2 -20464.318} C_VEL
LIN {X 0,Y 220.796,Z 278.482,A -85,B 0,C 180,E1 -20467.295,E2 -20467.295} C_VEL
LIN {X 0,Y 220.82,Z 278.479,A -85,B 0,C 180,E1 -20471.94,E2 -20471.94} C_VEL
LIN {X 0,Y 220.832,Z 278.478,A -85,B 0,C 180,E1 -20475.579,E2 -20475.579} C_VEL
LIN {X 0,Y 220.823,Z 278.478,A -85,B 0,C 180,E1 -20480.483,E2 -20480.483} C_VEL
LIN {X 0,Y 220.785,Z 278.483,A -85,B 0,C 180,E1 -20485.058,E2 -20485.058} C_VEL
LIN {X 0,Y 220.842,Z 278.477,A -85,B 0,C 180,E1 -20489.405,E2 -20489.405} C_VEL
LIN {X 0,Y 220.87,Z 278.47,A -85,B 0,C 180,E1 -20493.56,E2 -20493.56} C_VEL
LIN {X 0,Y 220.843,Z 278.475,A -85,B 0,C 180,E1 -20497.563,E2 -20497.563} C_VEL
LIN {X 0,Y 220.912,Z 278.468,A -85,B 0,C 180,E1 -20502.628,E2 -20502.628} C_VEL
LIN {X 0,Y 220.981,Z 278.459,A -85,B 0,C 180,E1 -20507.148,E2 -20507.148} C_VEL
LIN {X 0,Y 221.189,Z 278.429,A -85,B 0,C 180,E1 -20510.87,E2 -20510.87} C_VEL
LIN {X 0,Y 221.239,Z 278.428,A -85,B 0,C 180,E1 -20512.711,E2 -20512.711} C_VEL
LIN {X 0,Y 221.465,Z 278.372,A -85,B 0,C 180,E1 -20518.192,E2 -20518.192} C_VEL
LIN {X 0,Y 221.465,Z 278.395,A -85,B 0,C 180,E1 -20521.829,E2 -20521.829} C_VEL
LIN {X 0,Y 221.241,Z 278.426,A -85,B 0,C 180,E1 -20527.31,E2 -20527.31} C_VEL
LIN {X 0,Y 221.053,Z 278.449,A -85,B 0,C 180,E1 -20531.007,E2 -20531.007} C_VEL
LIN {X 0,Y 220.976,Z 278.459,A -85,B 0,C 180,E1 -20536.643,E2 -20536.643} C_VEL
LIN {X 0,Y 220.854,Z 278.474,A -85,B 0,C 180,E1 -20540.5,E2 -20540.5} C_VEL
LIN {X 0,Y 220.806,Z 278.48,A -85,B 0,C 180,E1 -20544.452,E2 -20544.452} C_VEL
LIN {X 0,Y 220.86,Z 278.476,A -85,B 0,C 180,E1 -20547.004,E2 -20547.004} C_VEL
LIN {X 0,Y 221.011,Z 279.977,A -85,B 0,C 180,E1 -20550.844,E2 -20550.844} C_VEL
LIN {X 0,Y 221.278,Z 281.772,A -85,B 0,C 180,E1 -20554.879,E2 -20554.879} C_VEL
LIN {X 0,Y 221.582,Z 283.998,A -85,B 0,C 180,E1 -20559.382,E2 -20559.382} C_VEL
LIN {X 0,Y 221.848,Z 286.107,A -85,B 0,C 180,E1 -20563.23,E2 -20563.23} C_VEL
LIN {X 0,Y 221.925,Z 288.197,A -85,B 0,C 180,E1 -20566.762,E2 -20566.762} C_VEL
LIN {X 0,Y 221.536,Z 290.695,A -85,B 0,C 180,E1 -20570.62,E2 -20570.62} C_VEL
LIN {X 0,Y 221.187,Z 292.223,A -85,B 0,C 180,E1 -20572.865,E2 -20572.865} C_VEL
LIN {X 0,Y 220.628,Z 294.545,A -85,B 0,C 180,E1 -20575.93,E2 -20575.93} C_VEL
LIN {X 0,Y 221.598,Z 297.769,A -85,B 0,C 180,E1 -20576.263,E2 -20576.263} C_VEL
LIN {X 0,Y 225.418,Z 309.856,A -85,B 0,C 180,E1 -20577.804,E2 -20577.804} C_VEL
LIN {X 0,Y 227.914,Z 320.42,A -85,B 0,C 180,E1 -20579.281,E2 -20579.281} C_VEL
LIN {X 0,Y 229.612,Z 331.29,A -85,B 0,C 180,E1 -20580.954,E2 -20580.954} C_VEL
LIN {X 0,Y 230.484,Z 340.754,A -85,B 0,C 180,E1 -20582.583,E2 -20582.583} C_VEL
LIN {X 0,Y 230.612,Z 349.751,A -85,B 0,C 180,E1 -20584.312,E2 -20584.312} C_VEL
LIN {X 0,Y 230.38,Z 352.937,A -85,B 0,C 180,E1 -20584.959,E2 -20584.959} C_VEL
LIN {X 0,Y 227.563,Z 363.653,A -85,B 0,C 180,E1 -20587.292,E2 -20587.292} C_VEL
LIN {X 0,Y 227.486,Z 363.942,A -85,B 0,C 180,E1 -20587.369,E2 -20587.369} C_VEL
LIN {X 0,Y 225.813,Z 368.035,A -85,B 0,C 180,E1 -20588.394,E2 -20588.394} C_VEL
LIN {X 0,Y 221.4,Z 374.108,A -85,B 0,C 180,E1 -20590.031,E2 -20590.031} C_VEL
LIN {X 0,Y 217.01,Z 379.7,A -85,B 0,C 180,E1 -20591.841,E2 -20591.841} C_VEL
LIN {X 0,Y 215.402,Z 382.705,A -85,B 0,C 180,E1 -20593.12,E2 -20593.12} C_VEL
LIN {X 0,Y 213.791,Z 387.813,A -85,B 0,C 180,E1 -20595.727,E2 -20595.727} C_VEL
LIN {X 0,Y 212.668,Z 392.146,A -85,B 0,C 180,E1 -20598.564,E2 -20598.564} C_VEL
LIN {X 0,Y 212.114,Z 394.517,A -85,B 0,C 180,E1 -20600.464,E2 -20600.464} C_VEL
LIN {X 0,Y 211.722,Z 396.321,A -85,B 0,C 180,E1 -20602.37,E2 -20602.37} C_VEL
LIN {X 0,Y 211.444,Z 398.778,A -85,B 0,C 180,E1 -20606.188,E2 -20606.188} C_VEL
LIN {X 0,Y 211.445,Z 399.372,A -85,B 0,C 180,E1 -20608.095,E2 -20608.095} C_VEL
LIN {X 0,Y 211.539,Z 399.53,A -85,B 0,C 180,E1 -20610,E2 -20610} C_VEL
LIN {X 0,Y 211.445,Z 399.372,A -85,B 0,C 180,E1 -20611.905,E2 -20611.905} C_VEL
LIN {X 0,Y 211.473,Z 398.57,A -85,B 0,C 180,E1 -20614.337,E2 -20614.337} C_VEL
LIN {X 0,Y 211.746,Z 396.321,A -85,B 0,C 180,E1 -20617.629,E2 -20617.629} C_VEL
LIN {X 0,Y 212.384,Z 393.365,A -85,B 0,C 180,E1 -20620.486,E2 -20620.486} C_VEL
LIN {X 0,Y 213.359,Z 389.369,A -85,B 0,C 180,E1 -20623.331,E2 -20623.331} C_VEL
LIN {X 0,Y 214.904,Z 384.236,A -85,B 0,C 180,E1 -20626.139,E2 -20626.139} C_VEL
LIN {X 0,Y 216.488,Z 378.971,A -85,B 0,C 180,E1 -20628.452,E2 -20628.452} C_VEL
LIN {X 0,Y 218.464,Z 372.654,A -85,B 0,C 180,E1 -20630.724,E2 -20630.724} C_VEL
LIN {X 0,Y 220.537,Z 365.069,A -85,B 0,C 180,E1 -20632.978,E2 -20632.978} C_VEL
LIN {X 0,Y 223.088,Z 355.93,A -85,B 0,C 180,E1 -20635.169,E2 -20635.169} C_VEL
LIN {X 0,Y 223.877,Z 352.722,A -85,B 0,C 180,E1 -20635.821,E2 -20635.821} C_VEL
LIN {X 0,Y 223.936,Z 344.406,A -85,B 0,C 180,E1 -20637.566,E2 -20637.566} C_VEL
LIN {X 0,Y 223.445,Z 335.851,A -85,B 0,C 180,E1 -20639.176,E2 -20639.176} C_VEL
LIN {X 0,Y 222.169,Z 325.707,A -85,B 0,C 180,E1 -20640.886,E2 -20640.886} C_VEL
LIN {X 0,Y 220.388,Z 316.496,A -85,B 0,C 180,E1 -20642.309,E2 -20642.309} C_VEL
LIN {X 0,Y 217.298,Z 305.001,A -85,B 0,C 180,E1 -20643.938,E2 -20643.938} C_VEL
LIN {X 0,Y 214.564,Z 297.266,A -85,B 0,C 180,E1 -20645.014,E2 -20645.014} C_VEL
LIN {X 0,Y 213.752,Z 294.201,A -85,B 0,C 180,E1 -20645.34,E2 -20645.34} C_VEL
LIN {X 0,Y 214.324,Z 292.001,A -85,B 0,C 180,E1 -20648.537,E2 -20648.537} C_VEL
LIN {X 0,Y 214.701,Z 290.299,A -85,B 0,C 180,E1 -20651.147,E2 -20651.147} C_VEL
LIN {X 0,Y 214.86,Z 288.604,A -85,B 0,C 180,E1 -20653.966,E2 -20653.966} C_VEL
LIN {X 0,Y 214.81,Z 287.096,A -85,B 0,C 180,E1 -20656.59,E2 -20656.59} C_VEL
LIN {X 0,Y 214.669,Z 285.745,A -85,B 0,C 180,E1 -20659.086,E2 -20659.086} C_VEL
LIN {X 0,Y 214.29,Z 283.409,A -85,B 0,C 180,E1 -20663.808,E2 -20663.808} C_VEL
LIN {X 0,Y 214.003,Z 281.276,A -85,B 0,C 180,E1 -20668.632,E2 -20668.632} C_VEL
LIN {X 0,Y 213.84,Z 279.725,A -85,B 0,C 180,E1 -20672.595,E2 -20672.595} C_VEL
LIN {X 0,Y 213.774,Z 279.363,A -85,B 0,C 180,E1 -20676.754,E2 -20676.754} C_VEL
LIN {X 0,Y 213.798,Z 279.356,A -85,B 0,C 180,E1 -20680.798,E2 -20680.798} C_VEL
LIN {X 0,Y 213.876,Z 279.344,A -85,B 0,C 180,E1 -20684.749,E2 -20684.749} C_VEL
LIN {X 0,Y 214.135,Z 279.311,A -85,B 0,C 180,E1 -20690.544,E2 -20690.544} C_VEL
LIN {X 0,Y 214.072,Z 279.319,A -85,B 0,C 180,E1 -20694.337,E2 -20694.337} C_VEL
LIN {X 0,Y 214.401,Z 279.275,A -85,B 0,C 180,E1 -20698.111,E2 -20698.111} C_VEL
LIN {X 0,Y 214.507,Z 279.25,A -85,B 0,C 180,E1 -20699.989,E2 -20699.989} C_VEL
LIN {X 0,Y 214.402,Z 279.25,A -85,B 0,C 180,E1 -20701.867,E2 -20701.867} C_VEL
LIN {X 0,Y 214.179,Z 279.307,A -85,B 0,C 180,E1 -20707.531,E2 -20707.531} C_VEL
LIN {X 0,Y 213.981,Z 279.329,A -85,B 0,C 180,E1 -20711.353,E2 -20711.353} C_VEL
LIN {X 0,Y 213.886,Z 279.337,A -85,B 0,C 180,E1 -20715.228,E2 -20715.228} C_VEL
LIN {X 0,Y 213.795,Z 279.349,A -85,B 0,C 180,E1 -20719.179,E2 -20719.179} C_VEL
LIN {X 0,Y 213.789,Z 279.353,A -85,B 0,C 180,E1 -20723.22,E2 -20723.22} C_VEL
LIN {X 0,Y 213.805,Z 279.352,A -85,B 0,C 180,E1 -20727.439,E2 -20727.439} C_VEL
LIN {X 0,Y 213.752,Z 279.358,A -85,B 0,C 180,E1 -20731.725,E2 -20731.725} C_VEL
LIN {X 0,Y 213.723,Z 279.362,A -85,B 0,C 180,E1 -20736.276,E2 -20736.276} C_VEL
LIN {X 0,Y 213.762,Z 279.358,A -85,B 0,C 180,E1 -20741.096,E2 -20741.096} C_VEL
LIN {X 0,Y 213.8,Z 279.353,A -85,B 0,C 180,E1 -20743.684,E2 -20743.684} C_VEL
LIN {X 0,Y 213.774,Z 279.358,A -85,B 0,C 180,E1 -20746.34,E2 -20746.34} C_VEL
LIN {X 0,Y 213.757,Z 279.357,A -85,B 0,C 180,E1 -20749.11,E2 -20749.11} C_VEL
LIN {X 0,Y 213.702,Z 279.367,A -85,B 0,C 180,E1 -20753.704,E2 -20753.704} C_VEL
LIN {X 0,Y 213.692,Z 279.368,A -85,B 0,C 180,E1 -20754.402,E2 -20754.402} C_VEL
LIN {X 0,Y 214.736,Z 282.268,A -85,B 0,C 180,E1 -20754.773,E2 -20754.773} C_VEL
LIN {X 0,Y 216.134,Z 284.425,A -85,B 0,C 180,E1 -20755.153,E2 -20755.153} C_VEL
LIN {X 0,Y 221.042,Z 293.46,A -85,B 0,C 180,E1 -20756.655,E2 -20756.655} C_VEL
LIN {X 0,Y 225.746,Z 303.73,A -85,B 0,C 180,E1 -20758.387,E2 -20758.387} C_VEL
LIN {X 0,Y 229.606,Z 314.175,A -85,B 0,C 180,E1 -20760.218,E2 -20760.218} C_VEL
LIN {X 0,Y 233.122,Z 323.944,A -85,B 0,C 180,E1 -20762.141,E2 -20762.141} C_VEL
LIN {X 0,Y 237.696,Z 333.313,A -85,B 0,C 180,E1 -20764.366,E2 -20764.366} C_VEL
LIN {X 0,Y 244.107,Z 343.051,A -85,B 0,C 180,E1 -20767.084,E2 -20767.084} C_VEL
LIN {X 0,Y 251.806,Z 351.961,A -85,B 0,C 180,E1 -20769.984,E2 -20769.984} C_VEL
LIN {X 0,Y 260.753,Z 360.246,A -85,B 0,C 180,E1 -20773.056,E2 -20773.056} C_VEL
LIN {X 0,Y 270.444,Z 367.692,A -85,B 0,C 180,E1 -20776.221,E2 -20776.221} C_VEL
LIN {X 0,Y 276.614,Z 371.942,A -85,B 0,C 180,E1 -20778.273,E2 -20778.273} C_VEL
LIN {X 0,Y 283.163,Z 376.205,A -85,B 0,C 180,E1 -20780.624,E2 -20780.624} C_VEL
LIN {X 0,Y 288.948,Z 379.751,A -85,B 0,C 180,E1 -20783.015,E2 -20783.015} C_VEL
LIN {X 0,Y 291.357,Z 381.474,A -85,B 0,C 180,E1 -20784.463,E2 -20784.463} C_VEL
LIN {X 0,Y 293.448,Z 382.793,A -85,B 0,C 180,E1 -20785.88,E2 -20785.88} C_VEL
LIN {X 0,Y 295.441,Z 383.755,A -85,B 0,C 180,E1 -20787.317,E2 -20787.317} C_VEL
LIN {X 0,Y 296.843,Z 384.279,A -85,B 0,C 180,E1 -20788.643,E2 -20788.643} C_VEL
LIN {X 0,Y 297.714,Z 384.454,A -85,B 0,C 180,E1 -20790,E2 -20790} C_VEL
LIN {X 0,Y 296.836,Z 384.28,A -85,B 0,C 180,E1 -20791.357,E2 -20791.357} C_VEL
LIN {X 0,Y 295.365,Z 383.729,A -85,B 0,C 180,E1 -20792.728,E2 -20792.728} C_VEL
LIN {X 0,Y 293.446,Z 382.792,A -85,B 0,C 180,E1 -20794.12,E2 -20794.12} C_VEL
LIN {X 0,Y 289.93,Z 380.407,A -85,B 0,C 180,E1 -20796.459,E2 -20796.459} C_VEL
LIN {X 0,Y 287.232,Z 378.718,A -85,B 0,C 180,E1 -20797.734,E2 -20797.734} C_VEL
LIN {X 0,Y 281.316,Z 374.998,A -85,B 0,C 180,E1 -20800.071,E2 -20800.071} C_VEL
LIN {X 0,Y 276.613,Z 371.942,A -85,B 0,C 180,E1 -20801.727,E2 -20801.727} C_VEL
LIN {X 0,Y 268.44,Z 366.273,A -85,B 0,C 180,E1 -20804.424,E2 -20804.424} C_VEL
LIN {X 0,Y 259.634,Z 359.266,A -85,B 0,C 180,E1 -20807.323,E2 -20807.323} C_VEL
LIN {X 0,Y 251.833,Z 351.92,A -85,B 0,C 180,E1 -20810.025,E2 -20810.025} C_VEL
LIN {X 0,Y 244.112,Z 343.037,A -85,B 0,C 180,E1 -20812.919,E2 -20812.919} C_VEL
LIN {X 0,Y 238.432,Z 334.592,A -85,B 0,C 180,E1 -20815.302,E2 -20815.302} C_VEL
